KUKA KRL program: MyProgram_148().src

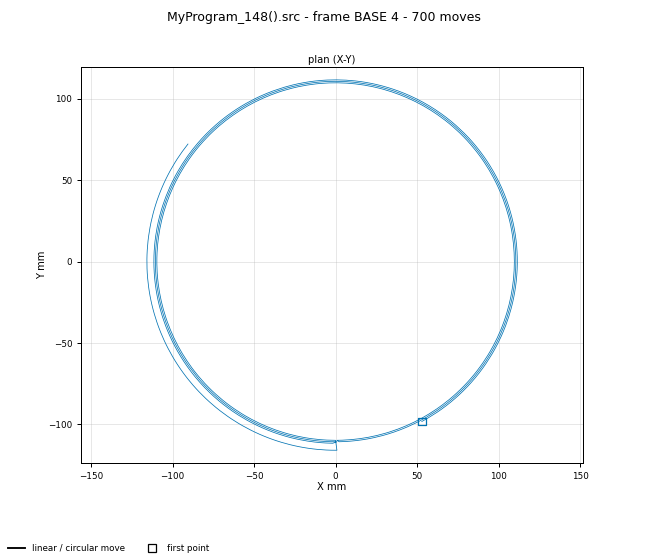
[picture p0: tool path of MyProgram_148().src in frame BASE 4, 700 of 700 moves have a stored position in this frame; points joined in program order, loops and branches not executed]
&ACCESS RVP
&REL 1
&PARAM TEMPLATE = C:\KRC\Roboter\Template\vorgabe
&PARAM EDITMASK = *
DEF MyProgram_148()
; ---- Setting reference (Base) ----
$BASE = BASE_DATA[4]

; --------------------------
; ---- Setting tool (TCP) ----
$TOOL = TOOL_DATA[3]
; --------------------------

$VEL.CP = VEL_APROX_PRINT
Startdeposition()
$VEL.CP = VEL_PRINT
LIN {X 52.9092,Y -98.1836,Z 116,A -65.1294,B 24.9503,C -1.6291,E1 25.0771,E2 510.9527} C_DIS
LIN {X 56.1114,Y -96.3909,Z 116,A -62.9664,B 24.9493,C -1.6449,E1 25.0824,E2 508.7589} C_DIS
LIN {X 62.3127,Y -92.5013,Z 116,A -59.4929,B 24.9496,C -1.6394,E1 25.0905,E2 505.3097} C_DIS
LIN {X 64.7563,Y -90.8071,Z 116,A -57.9766,B 24.9495,C -1.642,E1 25.094,E2 503.7925} C_DIS
LIN {X 67.8359,Y -88.5308,Z 116,A -55.9854,B 24.9491,C -1.6473,E1 25.0984,E2 501.7959} C_DIS
LIN {X 70.585,Y -86.3555,Z 116,A -54.1202,B 24.9487,C -1.6542,E1 25.1025,E2 499.9216} C_DIS
LIN {X 73.3349,Y -84.0315,Z 116,A -52.3931,B 24.9488,C -1.6529,E1 25.1062,E2 498.2042} C_DIS
LIN {X 75.9292,Y -81.6976,Z 116,A -50.5067,B 24.9483,C -1.6614,E1 25.1101,E2 496.3055} C_DIS
LIN {X 78.3692,Y -79.3573,Z 116,A -48.8923,B 24.9483,C -1.6601,E1 25.1133,E2 494.7009} C_DIS
LIN {X 80.9245,Y -76.7513,Z 116,A -47.0003,B 24.948,C -1.6655,E1 25.117,E2 492.8042} C_DIS
LIN {X 83.3621,Y -74.096,Z 116,A -45.0491,B 24.9474,C -1.6748,E1 25.1206,E2 490.8398} C_DIS
LIN {X 85.7734,Y -71.2898,Z 116,A -43.2959,B 24.9475,C -1.6731,E1 25.1238,E2 489.0986} C_DIS
LIN {X 87.8724,Y -68.6885,Z 116,A -41.4437,B 24.9469,C -1.6839,E1 25.127,E2 487.2296} C_DIS
LIN {X 90.2553,Y -65.5248,Z 116,A -39.4352,B 24.9466,C -1.6883,E1 25.1303,E2 485.2204} C_DIS
LIN {X 92.2402,Y -62.6984,Z 116,A -37.8546,B 24.9468,C -1.6844,E1 25.1328,E2 483.6567} C_DIS
LIN {X 95.8631,Y -57.0057,Z 116,A -34.2163,B 24.9457,C -1.7022,E1 25.1382,E2 479.9948} C_DIS
LIN {X 97.4564,Y -54.2363,Z 116,A -32.1233,B 24.9441,C -1.7278,E1 25.1412,E2 477.8523} C_DIS
LIN {X 99.4062,Y -50.5743,Z 116,A -30.4639,B 24.945,C -1.7125,E1 25.1432,E2 476.2379} C_DIS
LIN {X 101.6484,Y -45.9013,Z 116,A -27.9485,B 24.945,C -1.7138,E1 25.1462,E2 473.733} C_DIS
LIN {X 102.9872,Y -42.8163,Z 116,A -26.2004,B 24.9446,C -1.72,E1 25.1481,E2 471.9797} C_DIS
LIN {X 104.3967,Y -39.2519,Z 116,A -24.253,B 24.9442,C -1.7252,E1 25.1501,E2 470.031} C_DIS
LIN {X 105.5601,Y -36.0073,Z 116,A -22.4909,B 24.9439,C -1.7304,E1 25.1517,E2 468.2667} C_DIS
LIN {X 106.3439,Y -33.6253,Z 116,A -20.9984,B 24.943,C -1.7438,E1 25.153,E2 466.751} C_DIS
LIN {X 107.7745,Y -28.7076,Z 116,A -18.5694,B 24.943,C -1.7429,E1 25.1548,E2 464.338} C_DIS
LIN {X 108.7112,Y -24.9243,Z 116,A -16.7996,B 24.9433,C -1.7387,E1 25.1559,E2 462.5884} C_DIS
LIN {X 109.3364,Y -22.0232,Z 116,A -15.2816,B 24.943,C -1.7433,E1 25.1568,E2 461.0683} C_DIS
LIN {X 109.9232,Y -18.8799,Z 116,A -13.4529,B 24.9421,C -1.7571,E1 25.1577,E2 459.2177} C_DIS
LIN {X 110.4369,Y -15.5885,Z 116,A -11.7848,B 24.9419,C -1.7607,E1 25.1584,E2 457.551} C_DIS
LIN {X 110.8616,Y -12.2227,Z 116,A -10.0076,B 24.9414,C -1.768,E1 25.159,E2 455.7672} C_DIS
LIN {X 111.2013,Y -8.5827,Z 116,A -7.8213,B 24.9401,C -1.7883,E1 25.1595,E2 453.5459} C_DIS
LIN {X 111.4062,Y -5.3144,Z 116,A -6.3852,B 24.9405,C -1.7824,E1 25.1597,E2 452.1322} C_DIS
LIN {X 111.5251,Y -1.3818,Z 116,A -4.5343,B 24.9405,C -1.7812,E1 25.1597,E2 450.2953} C_DIS
LIN {X 111.4999,Y 2.7453,Z 116,A -1.9208,B 24.9385,C -1.8108,E1 25.1597,E2 447.6275} C_DIS
LIN {X 111.3508,Y 6.351,Z 116,A -0.5664,B 24.9397,C -1.7938,E1 25.1595,E2 446.3212} C_DIS
LIN {X 111.1521,Y 9.1985,Z 116,A 1.3678,B 24.9379,C -1.82,E1 25.159,E2 444.3366} C_DIS
LIN {X 110.7896,Y 12.8447,Z 116,A 2.7241,B 24.9391,C -1.8019,E1 25.1586,E2 443.0311} C_DIS
LIN {X 110.2953,Y 16.5677,Z 116,A 4.7378,B 24.9385,C -1.8119,E1 25.1578,E2 441.0057} C_DIS
LIN {X 109.7106,Y 20.0748,Z 116,A 6.5958,B 24.938,C -1.8191,E1 25.1569,E2 439.1416} C_DIS
LIN {X 108.9851,Y 23.6972,Z 116,A 8.3703,B 24.938,C -1.8194,E1 25.1559,E2 437.3767} C_DIS
LIN {X 108.1757,Y 27.161,Z 116,A 10.2711,B 24.9373,C -1.8284,E1 25.1546,E2 435.4655} C_DIS
LIN {X 107.3561,Y 30.2325,Z 116,A 11.7358,B 24.9375,C -1.8258,E1 25.1536,E2 434.0154} C_DIS
LIN {X 106.2715,Y 33.8515,Z 116,A 13.8167,B 24.9367,C -1.8381,E1 25.1518,E2 431.9175} C_DIS
LIN {X 105.0919,Y 37.3513,Z 116,A 16.2291,B 24.9346,C -1.8674,E1 25.1496,E2 429.4496} C_DIS
LIN {X 103.5813,Y 41.3594,Z 116,A 18.0483,B 24.9354,C -1.8564,E1 25.1477,E2 427.6663} C_DIS
LIN {X 101.9341,Y 45.2672,Z 116,A 20.0203,B 24.9356,C -1.8533,E1 25.1455,E2 425.7125} C_DIS
LIN {X 100.5925,Y 48.1713,Z 116,A 21.698,B 24.9352,C -1.8596,E1 25.1435,E2 424.029} C_DIS
LIN {X 98.7423,Y 51.8584,Z 116,A 23.6261,B 24.9354,C -1.8568,E1 25.1411,E2 422.1176} C_DIS
LIN {X 97.0537,Y 54.9566,Z 116,A 25.6699,B 24.9343,C -1.8722,E1 25.1383,E2 420.0482} C_DIS
LIN {X 94.5285,Y 59.1919,Z 116,A 28.0302,B 24.9343,C -1.8712,E1 25.1349,E2 417.7022} C_DIS
LIN {X 92.7016,Y 62.017,Z 116,A 29.8036,B 24.9339,C -1.8777,E1 25.1322,E2 415.9223} C_DIS
LIN {X 91.0092,Y 64.473,Z 116,A 31.3362,B 24.9336,C -1.8816,E1 25.1297,E2 414.388} C_DIS
LIN {X 88.7627,Y 67.5349,Z 116,A 33.5767,B 24.9324,C -1.8994,E1 25.1259,E2 412.1161} C_DIS
LIN {X 85.9589,Y 71.0665,Z 116,A 35.5596,B 24.933,C -1.89,E1 25.1225,E2 410.1646} C_DIS
LIN {X 83.7079,Y 73.7055,Z 116,A 37.3159,B 24.9328,C -1.893,E1 25.1192,E2 408.4092} C_DIS
LIN {X 81.6754,Y 75.9528,Z 116,A 39.3987,B 24.9309,C -1.9201,E1 25.1152,E2 406.2717} C_DIS
LIN {X 78.9056,Y 78.8264,Z 116,A 40.8065,B 24.9326,C -1.8958,E1 25.1125,E2 404.9272} C_DIS
LIN {X 73.6893,Y 83.722,Z 116,A 44.6367,B 24.9316,C -1.9102,E1 25.1047,E2 401.0785} C_DIS
LIN {X 70.7104,Y 86.2539,Z 116,A 46.6082,B 24.9314,C -1.9124,E1 25.1004,E2 399.1093} C_DIS
LIN {X 67.7988,Y 88.5593,Z 116,A 48.5399,B 24.9311,C -1.917,E1 25.0962,E2 397.174} C_DIS
LIN {X 64.6194,Y 90.9048,Z 116,A 50.7894,B 24.9302,C -1.9302,E1 25.091,E2 394.9011} C_DIS
LIN {X 60.8841,Y 93.4495,Z 116,A 52.8224,B 24.9308,C -1.9213,E1 25.0863,E2 392.896} C_DIS
LIN {X 57.336,Y 95.668,Z 116,A 55.1632,B 24.93,C -1.9329,E1 25.0807,E2 390.535} C_DIS
LIN {X 53.72,Y 97.7434,Z 116,A 57.238,B 24.93,C -1.933,E1 25.0757,E2 388.4661} C_DIS
LIN {X 49.7844,Y 99.8043,Z 116,A 59.6973,B 24.9292,C -1.9437,E1 25.0695,E2 385.9882} C_DIS
LIN {X 45.4869,Y 101.8351,Z 116,A 61.7418,B 24.9302,C -1.9293,E1 25.0644,E2 383.9829} C_DIS
LIN {X 42.4471,Y 103.1394,Z 116,A 63.4921,B 24.9299,C -1.9333,E1 25.0599,E2 382.2272} C_DIS
LIN {X 38.7978,Y 104.5678,Z 116,A 65.399,B 24.9301,C -1.9307,E1 25.055,E2 380.3308} C_DIS
LIN {X 35.1737,Y 105.8412,Z 116,A 67.4613,B 24.9297,C -1.9362,E1 25.0495,E2 378.2594} C_DIS
LIN {X 32.2727,Y 106.7609,Z 116,A 69.4841,B 24.9282,C -1.9572,E1 25.044,E2 376.1905} C_DIS
LIN {X 28.7542,Y 107.7619,Z 116,A 70.8582,B 24.9297,C -1.9368,E1 25.0404,E2 374.867} C_DIS
LIN {X 25.1913,Y 108.6495,Z 116,A 72.7621,B 24.9295,C -1.9386,E1 25.0352,E2 372.9615} C_DIS
LIN {X 22.2287,Y 109.2943,Z 116,A 74.4419,B 24.9291,C -1.9445,E1 25.0306,E2 371.2699} C_DIS
LIN {X 18.5918,Y 109.9713,Z 116,A 76.155,B 24.9296,C -1.9373,E1 25.0259,E2 369.5757} C_DIS
LIN {X 15.9494,Y 110.3857,Z 116,A 77.5464,B 24.9296,C -1.9384,E1 25.0221,E2 368.183} C_DIS
LIN {X 12.0058,Y 110.8843,Z 116,A 79.7842,B 24.9289,C -1.947,E1 25.0158,E2 365.9263} C_DIS
LIN {X 6.4381,Y 111.346,Z 116,A 82.5158,B 24.9293,C -1.9413,E1 25.0083,E2 363.2096} C_DIS
LIN {X 3.0813,Y 111.4896,Z 116,A 84.2013,B 24.9295,C -1.9395,E1 25.0036,E2 361.5289} C_DIS
LIN {X 0.6202,Y 111.5299,Z 116,A 85.7304,B 24.9287,C -1.9504,E1 24.9992,E2 359.9741} C_DIS
LIN {X -5.1396,Y 111.4137,Z 116,A 88.4976,B 24.9293,C -1.9414,E1 24.9916,E2 357.2277} C_DIS
LIN {X -8.4005,Y 111.216,Z 116,A 90.2558,B 24.9291,C -1.9441,E1 24.9867,E2 355.4626} C_DIS
LIN {X -12.4768,Y 110.8327,Z 116,A 92.6726,B 24.9283,C -1.956,E1 24.9799,E2 353.0162} C_DIS
LIN {X -15.8136,Y 110.405,Z 116,A 93.9929,B 24.9296,C -1.9379,E1 24.9763,E2 351.7375} C_DIS
LIN {X -19.4553,Y 109.8221,Z 116,A 95.9142,B 24.9296,C -1.9377,E1 24.971,E2 349.8151} C_DIS
LIN {X -23.038,Y 109.1281,Z 116,A 97.8293,B 24.9296,C -1.9377,E1 24.9658,E2 347.8977} C_DIS
LIN {X -26.4229,Y 108.3565,Z 116,A 99.5348,B 24.93,C -1.9329,E1 24.9612,E2 346.2014} C_DIS
LIN {X -29.291,Y 107.6169,Z 116,A 101.0996,B 24.93,C -1.9331,E1 24.9569,E2 344.6337} C_DIS
LIN {X -31.5254,Y 106.9836,Z 116,A 103.5992,B 24.9261,C -1.9857,E1 24.95,E2 342.0049} C_DIS
LIN {X -38.4898,Y 104.6801,Z 116,A 106.5973,B 24.9288,C -1.9489,E1 24.9423,E2 339.0881} C_DIS
LIN {X -42.1959,Y 103.2417,Z 116,A 108.6809,B 24.9288,C -1.9477,E1 24.9369,E2 337.0027} C_DIS
LIN {X -46.0009,Y 101.6034,Z 116,A 110.2767,B 24.9307,C -1.9229,E1 24.9329,E2 335.4621} C_DIS
LIN {X -49.297,Y 100.0459,Z 116,A 112.1442,B 24.9309,C -1.9197,E1 24.9283,E2 333.5974} C_DIS
LIN {X -54.9445,Y 97.061,Z 116,A 115.5039,B 24.9311,C -1.9172,E1 24.92,E2 330.2342} C_DIS
LIN {X -57.6585,Y 95.472,Z 116,A 117.0868,B 24.9314,C -1.9129,E1 24.9162,E2 328.6566} C_DIS
LIN {X -60.6647,Y 93.5914,Z 116,A 118.9691,B 24.9314,C -1.9118,E1 24.9118,E2 326.7708} C_DIS
LIN {X -63.5165,Y 91.6788,Z 116,A 120.8591,B 24.9314,C -1.9134,E1 24.9074,E2 324.8708} C_DIS
LIN {X -66.9482,Y 89.2034,Z 116,A 123.5372,B 24.9302,C -1.929,E1 24.9013,E2 322.1459} C_DIS
LIN {X -70.7502,Y 86.2217,Z 116,A 125.8474,B 24.9311,C -1.9166,E1 24.8964,E2 319.8565} C_DIS
LIN {X -73.7129,Y 83.7014,Z 116,A 127.3539,B 24.9329,C -1.8925,E1 24.8933,E2 318.4015} C_DIS
LIN {X -76.5079,Y 81.1534,Z 116,A 129.8759,B 24.9315,C -1.9109,E1 24.888,E2 315.8252} C_DIS
LIN {X -79.5478,Y 78.1763,Z 116,A 132.0811,B 24.9319,C -1.9063,E1 24.8837,E2 313.6216} C_DIS
LIN {X -82.5085,Y 75.0459,Z 116,A 133.7954,B 24.9337,C -1.8809,E1 24.8806,E2 311.9602} C_DIS
LIN {X -84.5818,Y 72.7012,Z 116,A 135.9859,B 24.9323,C -1.8998,E1 24.8765,E2 309.7147} C_DIS
LIN {X -87.4363,Y 69.2402,Z 116,A 137.8303,B 24.9341,C -1.8755,E1 24.8734,E2 307.9197} C_DIS
LIN {X -90.8086,Y 64.7542,Z 116,A 140.4061,B 24.9355,C -1.8556,E1 24.8692,E2 305.3789} C_DIS
LIN {X -94.0747,Y 59.9117,Z 116,A 143.6719,B 24.9353,C -1.8574,E1 24.8641,E2 302.0924} C_DIS
LIN {X -96.813,Y 55.3769,Z 116,A 146.2308,B 24.9363,C -1.8432,E1 24.8605,E2 299.5542} C_DIS
LIN {X -98.3015,Y 52.6919,Z 116,A 147.9315,B 24.9363,C -1.8434,E1 24.8582,E2 297.8441} C_DIS
LIN {X -100.3136,Y 48.7518,Z 116,A 150.216,B 24.9367,C -1.837,E1 24.8554,E2 295.5625} C_DIS
LIN {X -101.6068,Y 45.9935,Z 116,A 151.6526,B 24.9374,C -1.8273,E1 24.8537,E2 294.1411} C_DIS
LIN {X -104.1686,Y 39.8541,Z 116,A 155.2238,B 24.9377,C -1.8227,E1 24.8499,E2 290.5611} C_DIS
LIN {X -105.2317,Y 36.9541,Z 116,A 156.6956,B 24.9384,C -1.8133,E1 24.8485,E2 289.1033} C_DIS
LIN {X -106.0707,Y 34.4723,Z 116,A 158.7014,B 24.9369,C -1.8347,E1 24.8468,E2 287.0348} C_DIS
LIN {X -107.263,Y 30.561,Z 116,A 159.9553,B 24.9396,C -1.7952,E1 24.8459,E2 285.8681} C_DIS
LIN {X -108.04,Y 27.6889,Z 116,A 162.1523,B 24.9382,C -1.8162,E1 24.8443,E2 283.6082} C_DIS
LIN {X -108.826,Y 24.4269,Z 116,A 163.447,B 24.9397,C -1.794,E1 24.8435,E2 282.3589} C_DIS
LIN {X -109.5487,Y 20.9374,Z 116,A 166.1596,B 24.9377,C -1.8225,E1 24.842,E2 279.5622} C_DIS
LIN {X -110.3857,Y 15.9494,Z 116,A 168.0257,B 24.9403,C -1.7854,E1 24.8413,E2 277.7733} C_DIS
LIN {X -110.8645,Y 12.1948,Z 116,A 170.0214,B 24.9405,C -1.7811,E1 24.8406,E2 275.7761} C_DIS
LIN {X -111.1664,Y 9.0196,Z 116,A 171.5106,B 24.9413,C -1.77,E1 24.8402,E2 274.3043} C_DIS
LIN {X -111.3505,Y 6.3572,Z 116,A 172.8897,B 24.9416,C -1.7659,E1 24.84,E2 272.9268} C_DIS
LIN {X -111.4802,Y 3.3861,Z 116,A 174.5077,B 24.9416,C -1.7644,E1 24.8398,E2 271.3026} C_DIS
LIN {X -111.5316,Y -0.2035,Z 116,A 176.3564,B 24.942,C -1.7586,E1 24.8398,E2 269.4566} C_DIS
LIN {X -111.4807,Y -3.3722,Z 116,A 178.0458,B 24.9422,C -1.7557,E1 24.8399,E2 267.7639} C_DIS
LIN {X -111.3074,Y -7.0828,Z 116,A -179.9817,B 24.9425,C -1.752,E1 24.8402,E2 265.7883} C_DIS
LIN {X -110.9839,Y -11.0543,Z 116,A -178.0528,B 24.9432,C -1.7408,E1 24.8407,E2 263.8745} C_DIS
LIN {X -110.6319,Y -14.1394,Z 116,A -176.3798,B 24.9433,C -1.7388,E1 24.8413,E2 262.1964} C_DIS
LIN {X -110.1255,Y -17.6658,Z 116,A -174.4928,B 24.9436,C -1.7352,E1 24.8421,E2 260.3068} C_DIS
LIN {X -109.5137,Y -21.12,Z 116,A -172.7188,B 24.944,C -1.7284,E1 24.843,E2 258.5384} C_DIS
LIN {X -108.9187,Y -24.0018,Z 116,A -170.7974,B 24.9433,C -1.7397,E1 24.8441,E2 256.5787} C_DIS
LIN {X -108.1112,Y -27.4119,Z 116,A -169.4795,B 24.9449,C -1.7153,E1 24.845,E2 255.3114} C_DIS
LIN {X -106.7177,Y -32.4191,Z 116,A -166.7876,B 24.9453,C -1.7079,E1 24.8471,E2 252.6215} C_DIS
LIN {X -105.8504,Y -35.1463,Z 116,A -165.3312,B 24.9457,C -1.7029,E1 24.8483,E2 251.1686} C_DIS
LIN {X -104.284,Y -39.5494,Z 116,A -162.8738,B 24.946,C -1.698,E1 24.8507,E2 248.7091} C_DIS
LIN {X -103.0393,Y -42.6919,Z 116,A -161.0095,B 24.946,C -1.698,E1 24.8526,E2 246.8346} C_DIS
LIN {X -101.7991,Y -45.5668,Z 116,A -159.4265,B 24.9463,C -1.6923,E1 24.8544,E2 245.2562} C_DIS
LIN {X -100.3926,Y -48.5875,Z 116,A -157.7871,B 24.9468,C -1.6846,E1 24.8563,E2 243.6263} C_DIS
LIN {X -98.5083,Y -52.3026,Z 116,A -155.6007,B 24.9471,C -1.6805,E1 24.8592,E2 241.4381} C_DIS
LIN {X -97.1042,Y -54.8671,Z 116,A -153.8534,B 24.9467,C -1.6861,E1 24.8616,E2 239.6682} C_DIS
LIN {X -94.9548,Y -58.5095,Z 116,A -151.8064,B 24.9474,C -1.6753,E1 24.8645,E2 237.6364} C_DIS
LIN {X -93.0405,Y -61.5044,Z 116,A -150.0365,B 24.9478,C -1.6683,E1 24.8672,E2 235.8742} C_DIS
LIN {X -90.9636,Y -64.537,Z 116,A -148.186,B 24.9482,C -1.662,E1 24.8701,E2 234.0296} C_DIS
LIN {X -88.3938,Y -68.0134,Z 116,A -145.5244,B 24.9475,C -1.6742,E1 24.8747,E2 231.3262} C_DIS
LIN {X -86.2167,Y -70.7563,Z 116,A -144.0253,B 24.9485,C -1.6579,E1 24.8773,E2 229.8591} C_DIS
LIN {X -83.5848,Y -73.8464,Z 116,A -141.7264,B 24.9483,C -1.6617,E1 24.8815,E2 227.5407} C_DIS
LIN {X -80.3251,Y -77.3769,Z 116,A -139.5713,B 24.9494,C -1.6436,E1 24.8856,E2 225.4192} C_DIS
LIN {X -77.0941,Y -80.5977,Z 116,A -137.0655,B 24.9493,C -1.6452,E1 24.8906,E2 222.8991} C_DIS
LIN {X -74.3744,Y -83.1129,Z 116,A -135.3031,B 24.9499,C -1.6357,E1 24.8942,E2 221.1523} C_DIS
LIN {X -71.6856,Y -85.4445,Z 116,A -133.3821,B 24.9499,C -1.6359,E1 24.8983,E2 219.2234} C_DIS
LIN {X -69.227,Y -87.4468,Z 116,A -131.7489,B 24.95,C -1.6331,E1 24.9019,E2 217.5908} C_DIS
LIN {X -65.9884,Y -89.9158,Z 116,A -129.6715,B 24.9503,C -1.6288,E1 24.9065,E2 215.5162} C_DIS
LIN {X -63.0004,Y -92.0357,Z 116,A -127.7385,B 24.9503,C -1.6277,E1 24.911,E2 213.5792} C_DIS
LIN {X -59.5862,Y -94.2822,Z 116,A -125.4209,B 24.95,C -1.6333,E1 24.9165,E2 211.2407} C_DIS
LIN {X -54.3465,Y -97.3949,Z 116,A -122.5967,B 24.9511,C -1.6162,E1 24.9232,E2 208.4487} C_DIS
LIN {X -52.1961,Y -98.5644,Z 116,A -120.9552,B 24.9502,C -1.6304,E1 24.9273,E2 206.7689} C_DIS
LIN {X -48.1302,Y -100.6122,Z 116,A -118.9814,B 24.9513,C -1.6124,E1 24.9322,E2 204.8326} C_DIS
LIN {X -45.0177,Y -102.0439,Z 116,A -117.1605,B 24.9513,C -1.613,E1 24.9368,E2 203.0062} C_DIS
LIN {X -41.9734,Y -103.3322,Z 116,A -115.5832,B 24.9517,C -1.6062,E1 24.9409,E2 201.4413} C_DIS
LIN {X -38.2833,Y -104.7554,Z 116,A -113.4849,B 24.9517,C -1.6071,E1 24.9464,E2 199.3366} C_DIS
LIN {X -35.4239,Y -105.7568,Z 116,A -111.5717,B 24.9508,C -1.6207,E1 24.9515,E2 197.3873} C_DIS
LIN {X -30.6504,Y -107.2377,Z 116,A -109.3204,B 24.9517,C -1.6056,E1 24.9575,E2 195.1681} C_DIS
LIN {X -27.1861,Y -108.1692,Z 116,A -107.5707,B 24.952,C -1.6006,E1 24.9622,E2 193.4278} C_DIS
LIN {X -23.0365,Y -109.1284,Z 116,A -105.2378,B 24.9517,C -1.6056,E1 24.9686,E2 191.08} C_DIS
LIN {X -19.6611,Y -109.7851,Z 116,A -103.5339,B 24.9519,C -1.6024,E1 24.9732,E2 189.3821} C_DIS
LIN {X -17.1552,Y -110.2044,Z 116,A -102.0814,B 24.9515,C -1.6082,E1 24.9773,E2 187.9142} C_DIS
LIN {X -12.8611,Y -110.7877,Z 116,A -99.4591,B 24.9505,C -1.6248,E1 24.9847,E2 185.251} C_DIS
LIN {X -8.9519,Y -111.1718,Z 116,A -97.9302,B 24.9518,C -1.6037,E1 24.9888,E2 183.7712} C_DIS
LIN {X -6.097,Y -111.3649,Z 116,A -96.224,B 24.9512,C -1.6139,E1 24.9936,E2 182.0404} C_DIS
LIN {X -1.7181,Y -111.5189,Z 116,A -93.6675,B 24.9504,C -1.6275,E1 25.0009,E2 179.4515} C_DIS
LIN {X -1.7181,Y -111.5189,Z 116,A -93.6675,B 24.9504,C -1.6275,E1 25.0009,E2 179.4515} C_DIS
Enddeposition()
LIN {X 0.7946,Y -110.6158,Z 116,A -93.2714,B 24.9517,C -1.6052,E1 25.0018,E2 179.1083} C_DIS
Startdeposition()
$VEL.CP = VEL_PRINT
LIN {X -2.6442,Y -110.5946,Z 116,A -95.4467,B 24.9527,C -1.5881,E1 24.9956,E2 181.3241} C_DIS
LIN {X -6.5349,Y -110.4321,Z 116,A -97.5104,B 24.9529,C -1.586,E1 24.9898,E2 183.3933} C_DIS
LIN {X -9.5144,Y -110.2165,Z 116,A -99.3021,B 24.9535,C -1.5759,E1 24.9848,E2 185.2098} C_DIS
LIN {X -12.7964,Y -109.8819,Z 116,A -100.7721,B 24.9529,C -1.586,E1 24.9808,E2 186.6567} C_DIS
LIN {X -15.973,Y -109.466,Z 116,A -102.4709,B 24.9529,C -1.5847,E1 24.9761,E2 188.3599} C_DIS
LIN {X -19.2037,Y -108.9456,Z 116,A -103.9916,B 24.9525,C -1.5924,E1 24.9719,E2 189.8637} C_DIS
LIN {X -21.3846,Y -108.539,Z 116,A -105.2338,B 24.9527,C -1.589,E1 24.9685,E2 191.1153} C_DIS
LIN {X -23.5267,Y -108.0938,Z 116,A -106.4605,B 24.9529,C -1.5857,E1 24.9651,E2 192.3515} C_DIS
LIN {X -26.055,Y -107.5125,Z 116,A -107.7487,B 24.9527,C -1.5887,E1 24.9616,E2 193.6343} C_DIS
LIN {X -29.519,Y -106.6154,Z 116,A -109.5858,B 24.9527,C -1.5904,E1 24.9567,E2 195.47} C_DIS
LIN {X -31.9801,Y -105.9025,Z 116,A -111.4499,B 24.9538,C -1.5696,E1 24.9515,E2 197.3869} C_DIS
LIN {X -35.3248,Y -104.8329,Z 116,A -112.8332,B 24.9527,C -1.5887,E1 24.948,E2 198.7273} C_DIS
LIN {X -39.5172,Y -103.3262,Z 116,A -115.1086,B 24.9525,C -1.5921,E1 24.942,E2 200.9993} C_DIS
LIN {X -42.1139,Y -102.2956,Z 116,A -116.4787,B 24.9522,C -1.5966,E1 24.9385,E2 202.3616} C_DIS
LIN {X -45.0316,Y -101.0453,Z 116,A -118.0904,B 24.952,C -1.5997,E1 24.9344,E2 203.9697} C_DIS
LIN {X -47.1371,Y -100.0806,Z 116,A -119.3351,B 24.952,C -1.5993,E1 24.9312,E2 205.2186} C_DIS
LIN {X -49.1035,Y -99.1293,Z 116,A -120.4083,B 24.9519,C -1.603,E1 24.9285,E2 206.2857} C_DIS
LIN {X -52.1502,Y -97.5633,Z 116,A -122.269,B 24.9519,C -1.6018,E1 24.9239,E2 208.1544} C_DIS
LIN {X -55.258,Y -95.835,Z 116,A -124.1893,B 24.9519,C -1.6013,E1 24.9192,E2 210.0816} C_DIS
LIN {X -58.5749,Y -93.8444,Z 116,A -126.2251,B 24.9519,C -1.603,E1 24.9144,E2 212.1196} C_DIS
LIN {X -61.4116,Y -92.0151,Z 116,A -127.8814,B 24.9515,C -1.6094,E1 24.9105,E2 213.7661} C_DIS
LIN {X -64.1862,Y -90.0995,Z 116,A -129.7428,B 24.9515,C -1.6078,E1 24.9062,E2 215.6377} C_DIS
LIN {X -67.0583,Y -87.9847,Z 116,A -131.6136,B 24.9515,C -1.6101,E1 24.9021,E2 217.5097} C_DIS
LIN {X -69.7861,Y -85.8354,Z 116,A -133.3515,B 24.9511,C -1.6158,E1 24.8983,E2 219.2404} C_DIS
LIN {X -72.77,Y -83.3205,Z 116,A -135.3311,B 24.9507,C -1.6214,E1 24.8941,E2 221.2145} C_DIS
LIN {X -75.0304,Y -81.2916,Z 116,A -136.9337,B 24.9507,C -1.6234,E1 24.8908,E2 222.8188} C_DIS
LIN {X -77.8122,Y -78.6324,Z 116,A -138.945,B 24.9504,C -1.6269,E1 24.8867,E2 224.8301} C_DIS
LIN {X -80.025,Y -76.3811,Z 116,A -140.7607,B 24.9506,C -1.6233,E1 24.8832,E2 226.6621} C_DIS
LIN {X -82.6641,Y -73.5157,Z 116,A -142.5618,B 24.9498,C -1.6363,E1 24.8799,E2 228.4403} C_DIS
LIN {X -84.5753,Y -71.3101,Z 116,A -144.2654,B 24.9501,C -1.6323,E1 24.8767,E2 230.1611} C_DIS
LIN {X -89.8204,Y -64.5774,Z 116,A -148.4081,B 24.9487,C -1.6539,E1 24.8698,E2 234.2722} C_DIS
LIN {X -91.7647,Y -61.7827,Z 116,A -150.2724,B 24.9487,C -1.6544,E1 24.8668,E2 236.1443} C_DIS
LIN {X -93.4706,Y -59.1732,Z 116,A -151.9311,B 24.9486,C -1.6569,E1 24.8643,E2 237.8055} C_DIS
LIN {X -94.9201,Y -56.8183,Z 116,A -153.5828,B 24.9488,C -1.6523,E1 24.8618,E2 239.4767} C_DIS
LIN {X -96.9005,Y -53.3712,Z 116,A -155.6331,B 24.9485,C -1.6582,E1 24.859,E2 241.5237} C_DIS
LIN {X -98.55,Y -50.2563,Z 116,A -157.413,B 24.948,C -1.6651,E1 24.8568,E2 243.2968} C_DIS
LIN {X -100.3145,Y -46.6345,Z 116,A -159.4848,B 24.9476,C -1.6716,E1 24.8543,E2 245.3644} C_DIS
LIN {X -101.589,Y -43.7911,Z 116,A -160.9886,B 24.9471,C -1.6804,E1 24.8526,E2 246.8554} C_DIS
LIN {X -102.6665,Y -41.2027,Z 116,A -162.6467,B 24.9473,C -1.6768,E1 24.8508,E2 248.5314} C_DIS
LIN {X -104.1452,Y -37.309,Z 116,A -164.8304,B 24.947,C -1.6821,E1 24.8487,E2 250.7145} C_DIS
LIN {X -105.4494,Y -33.4457,Z 116,A -166.7619,B 24.9461,C -1.6954,E1 24.847,E2 252.6255} C_DIS
LIN {X -106.7136,Y -29.1561,Z 116,A -169.2007,B 24.946,C -1.6978,E1 24.8452,E2 255.0727} C_DIS
LIN {X -107.5482,Y -25.9087,Z 116,A -171.1503,B 24.9462,C -1.6951,E1 24.8438,E2 257.0401} C_DIS
LIN {X -108.4813,Y -21.6779,Z 116,A -173.3381,B 24.9456,C -1.7043,E1 24.8426,E2 259.219} C_DIS
LIN {X -109.2258,Y -17.5477,Z 116,A -175.2833,B 24.9446,C -1.7198,E1 24.8417,E2 261.1388} C_DIS
LIN {X -109.557,Y -15.3326,Z 116,A -176.4591,B 24.9444,C -1.7229,E1 24.8412,E2 262.3141} C_DIS
LIN {X -109.9712,Y -12.0151,Z 116,A -178.3434,B 24.9444,C -1.7226,E1 24.8406,E2 264.2103} C_DIS
LIN {X -110.2825,Y -8.6922,Z 116,A 179.9375,B 24.944,C -1.7286,E1 24.8402,E2 265.9256} C_DIS
LIN {X -110.4869,Y -5.5449,Z 116,A 178.4055,B 24.9434,C -1.7376,E1 24.8399,E2 267.4451} C_DIS
LIN {X -110.6035,Y -2.1578,Z 116,A 176.5375,B 24.9434,C -1.7391,E1 24.8398,E2 269.321} C_DIS
LIN {X -110.6116,Y 1.7189,Z 116,A 174.537,B 24.9429,C -1.7459,E1 24.8398,E2 271.3173} C_DIS
LIN {X -110.5029,Y 5.2045,Z 116,A 172.8221,B 24.9423,C -1.7552,E1 24.84,E2 273.0204} C_DIS
LIN {X -110.359,Y 7.6624,Z 116,A 171.3894,B 24.9423,C -1.7534,E1 24.8403,E2 274.4659} C_DIS
LIN {X -110.0288,Y 11.4645,Z 116,A 169.4518,B 24.9419,C -1.7613,E1 24.8408,E2 276.3963} C_DIS
LIN {X -109.5688,Y 15.2496,Z 116,A 166.3322,B 24.9442,C -1.725,E1 24.842,E2 279.6211} C_DIS
LIN {X -108.4938,Y 21.617,Z 116,A 164.1829,B 24.9406,C -1.7803,E1 24.8431,E2 281.6512} C_DIS
LIN {X -107.8858,Y 24.467,Z 116,A 162.0703,B 24.9418,C -1.7625,E1 24.8444,E2 283.8187} C_DIS
LIN {X -106.9715,Y 28.2015,Z 116,A 160.6439,B 24.9399,C -1.79,E1 24.8453,E2 285.1877} C_DIS
LIN {X -105.5341,Y 33.1742,Z 116,A 157.9865,B 24.9393,C -1.7995,E1 24.8474,E2 287.8381} C_DIS
LIN {X -104.5999,Y 36.0147,Z 116,A 156.2336,B 24.9395,C -1.7966,E1 24.849,E2 289.6078} C_DIS
LIN {X -103.2432,Y 39.7363,Z 116,A 154.1729,B 24.9391,C -1.8026,E1 24.851,E2 291.6657} C_DIS
LIN {X -101.5884,Y 43.7924,Z 116,A 152.1388,B 24.938,C -1.8185,E1 24.8532,E2 293.6732} C_DIS
LIN {X -100.4942,Y 46.2484,Z 116,A 150.4967,B 24.9384,C -1.8133,E1 24.8551,E2 295.3369} C_DIS
LIN {X -98.822,Y 49.7236,Z 116,A 148.3895,B 24.9382,C -1.8151,E1 24.8577,E2 297.4511} C_DIS
LIN {X -96.8267,Y 53.5033,Z 116,A 146.4794,B 24.937,C -1.8331,E1 24.8602,E2 299.3282} C_DIS
LIN {X -95.8824,Y 55.1757,Z 116,A 145.326,B 24.9372,C -1.83,E1 24.8618,E2 300.495} C_DIS
LIN {X -93.0955,Y 59.758,Z 116,A 142.8311,B 24.9359,C -1.8488,E1 24.8654,E2 302.958} C_DIS
LIN {X -91.647,Y 61.9565,Z 116,A 141.2159,B 24.9363,C -1.843,E1 24.8679,E2 304.5952} C_DIS
LIN {X -90.0404,Y 64.269,Z 116,A 139.0083,B 24.938,C -1.8186,E1 24.8716,E2 306.8716} C_DIS
LIN {X -87.3152,Y 67.9271,Z 116,A 137.3178,B 24.9358,C -1.8504,E1 24.8744,E2 308.4944} C_DIS
LIN {X -83.4721,Y 72.5964,Z 116,A 134.4396,B 24.9346,C -1.8684,E1 24.8795,E2 311.343} C_DIS
LIN {X -79.0901,Y 77.3489,Z 116,A 129.9716,B 24.937,C -1.834,E1 24.8882,E2 315.9125} C_DIS
LIN {X -75.4466,Y 80.9062,Z 116,A 128.2004,B 24.9342,C -1.8733,E1 24.8916,E2 317.5974} C_DIS
LIN {X -70.4463,Y 85.2949,Z 116,A 124.3381,B 24.9348,C -1.865,E1 24.8999,E2 321.4943} C_DIS
LIN {X -65.9354,Y 88.8296,Z 116,A 121.2904,B 24.9346,C -1.8682,E1 24.9067,E2 324.5454} C_DIS
LIN {X -63.2972,Y 90.7264,Z 116,A 120.172,B 24.9328,C -1.8935,E1 24.9091,E2 325.6074} C_DIS
LIN {X -60.8772,Y 92.3674,Z 116,A 118.4654,B 24.9331,C -1.889,E1 24.9131,E2 327.3304} C_DIS
LIN {X -58.4459,Y 93.9249,Z 116,A 116.9407,B 24.933,C -1.8907,E1 24.9167,E2 328.856} C_DIS
LIN {X -55.0438,Y 95.9582,Z 116,A 114.9108,B 24.9327,C -1.8953,E1 24.9216,E2 330.8809} C_DIS
LIN {X -51.2917,Y 98.0154,Z 116,A 112.8086,B 24.9321,C -1.9036,E1 24.9267,E2 332.9694} C_DIS
LIN {X -48.5101,Y 99.4233,Z 116,A 111.1536,B 24.932,C -1.9046,E1 24.9308,E2 334.6265} C_DIS
LIN {X -46.0536,Y 100.5847,Z 116,A 108.9137,B 24.9342,C -1.8742,E1 24.9367,E2 336.9442} C_DIS
LIN {X -41.711,Y 102.4596,Z 116,A 107.5962,B 24.9307,C -1.9222,E1 24.9399,E2 338.1505} C_DIS
LIN {X -39.5776,Y 103.3033,Z 116,A 105.9649,B 24.9319,C -1.9062,E1 24.9442,E2 339.8233} C_DIS
LIN {X -34.6704,Y 105.0516,Z 116,A 102.9692,B 24.9325,C -1.8979,E1 24.9522,E2 342.8447} C_DIS
LIN {X -29.2761,Y 106.6812,Z 116,A 100.5666,B 24.9308,C -1.9216,E1 24.9585,E2 345.1949} C_DIS
LIN {X -26.3675,Y 107.4363,Z 116,A 98.884,B 24.931,C -1.9181,E1 24.963,E2 346.8883} C_DIS
LIN {X -23.4553,Y 108.1094,Z 116,A 97.3098,B 24.931,C -1.9184,E1 24.9673,E2 348.4637} C_DIS
LIN {X -20.8527,Y 108.6414,Z 116,A 95.9727,B 24.9308,C -1.9211,E1 24.971,E2 349.7959} C_DIS
LIN {X -17.5603,Y 109.2239,Z 116,A 94.2367,B 24.9308,C -1.9222,E1 24.9758,E2 351.5311} C_DIS
LIN {X -13.6053,Y 109.7864,Z 116,A 91.9483,B 24.9313,C -1.9146,E1 24.9821,E2 353.8391} C_DIS
LIN {X -9.5612,Y 110.2122,Z 116,A 90.0651,B 24.9306,C -1.9247,E1 24.9873,E2 355.6994} C_DIS
LIN {X -6.5104,Y 110.4335,Z 116,A 88.3784,B 24.9308,C -1.9212,E1 24.992,E2 357.395} C_DIS
LIN {X -3.006,Y 110.5843,Z 116,A 86.545,B 24.9308,C -1.9211,E1 24.9972,E2 359.2289} C_DIS
LIN {X -0.2802,Y 110.6249,Z 116,A 85.1309,B 24.9308,C -1.9213,E1 25.0011,E2 360.6425} C_DIS
LIN {X 3.1623,Y 110.5795,Z 116,A 83.2783,B 24.931,C -1.9187,E1 25.0063,E2 362.501} C_DIS
LIN {X 6.9926,Y 110.4043,Z 116,A 81.3058,B 24.931,C -1.9193,E1 25.0118,E2 364.4714} C_DIS
LIN {X 11.0021,Y 110.0773,Z 116,A 79.4557,B 24.9303,C -1.9287,E1 25.0169,E2 366.2981} C_DIS
LIN {X 14.1649,Y 109.7139,Z 116,A 77.6114,B 24.9309,C -1.9203,E1 25.022,E2 368.1609} C_DIS
LIN {X 17.3527,Y 109.256,Z 116,A 76.0891,B 24.9305,C -1.9258,E1 25.0262,E2 369.6687} C_DIS
LIN {X 19.7772,Y 108.8425,Z 116,A 74.6396,B 24.931,C -1.9181,E1 25.0302,E2 371.1349} C_DIS
LIN {X 23.7373,Y 108.0479,Z 116,A 72.6248,B 24.9309,C -1.9203,E1 25.0357,E2 373.142} C_DIS
LIN {X 26.6627,Y 107.3643,Z 116,A 71.102,B 24.9309,C -1.9208,E1 25.0398,E2 374.6615} C_DIS
LIN {X 32.1205,Y 105.8607,Z 116,A 68.1593,B 24.931,C -1.9183,E1 25.0478,E2 377.6052} C_DIS
LIN {X 36.0617,Y 104.5834,Z 116,A 66.06,B 24.931,C -1.9184,E1 25.0533,E2 379.7001} C_DIS
LIN {X 38.6032,Y 103.6723,Z 116,A 64.7124,B 24.931,C -1.9193,E1 25.0568,E2 381.0429} C_DIS
LIN {X 40.6005,Y 102.9048,Z 116,A 63.5215,B 24.9313,C -1.9147,E1 25.0599,E2 382.242} C_DIS
LIN {X 43.5913,Y 101.6761,Z 116,A 61.9088,B 24.9313,C -1.9155,E1 25.0641,E2 383.8491} C_DIS
LIN {X 45.586,Y 100.7954,Z 116,A 60.6139,B 24.9318,C -1.9072,E1 25.0674,E2 385.1603} C_DIS
LIN {X 48.9503,Y 99.2053,Z 116,A 59.0717,B 24.9308,C -1.9212,E1 25.0712,E2 386.6654} C_DIS
LIN {X 51.077,Y 98.1285,Z 116,A 57.2285,B 24.9328,C -1.8938,E1 25.0759,E2 388.5685} C_DIS
LIN {X 55.3563,Y 95.7786,Z 116,A 55.1536,B 24.9316,C -1.9095,E1 25.0809,E2 390.6001} C_DIS
LIN {X 57.9023,Y 94.2623,Z 116,A 53.5737,B 24.932,C -1.9052,E1 25.0847,E2 392.1852} C_DIS
LIN {X 59.9967,Y 92.9422,Z 116,A 52.3407,B 24.932,C -1.9053,E1 25.0876,E2 393.4139} C_DIS
LIN {X 62.5047,Y 91.2758,Z 116,A 50.6446,B 24.9325,C -1.8969,E1 25.0915,E2 395.1243} C_DIS
LIN {X 65.2952,Y 89.299,Z 116,A 48.9091,B 24.9327,C -1.8953,E1 25.0954,E2 396.8573} C_DIS
LIN {X 68.3499,Y 86.9837,Z 116,A 46.9201,B 24.9329,C -1.8916,E1 25.0999,E2 398.8479} C_DIS
LIN {X 70.9145,Y 84.9058,Z 116,A 45.2638,B 24.9329,C -1.8906,E1 25.1034,E2 400.5002} C_DIS
LIN {X 73.4309,Y 82.74,Z 116,A 43.3584,B 24.9338,C -1.8792,E1 25.1075,E2 402.4251} C_DIS
LIN {X 76.4536,Y 79.9551,Z 116,A 41.3341,B 24.9338,C -1.8792,E1 25.1116,E2 404.4409} C_DIS
LIN {X 78.7151,Y 77.7285,Z 116,A 39.6124,B 24.9343,C -1.8723,E1 25.115,E2 406.1716} C_DIS
LIN {X 81.4654,Y 74.8409,Z 116,A 37.7115,B 24.9341,C -1.8749,E1 25.1186,E2 408.0582} C_DIS
LIN {X 83.4668,Y 72.6025,Z 116,A 36.1044,B 24.9345,C -1.869,E1 25.1216,E2 409.6718} C_DIS
LIN {X 85.8055,Y 69.823,Z 116,A 34.2828,B 24.9346,C -1.8672,E1 25.1248,E2 411.4895} C_DIS
LIN {X 88.0407,Y 66.9856,Z 116,A 32.4947,B 24.9347,C -1.8662,E1 25.1278,E2 413.2715} C_DIS
LIN {X 90.3627,Y 63.8173,Z 116,A 30.2523,B 24.9357,C -1.852,E1 25.1315,E2 415.5365} C_DIS
LIN {X 92.7904,Y 60.2333,Z 116,A 28.294,B 24.9352,C -1.8586,E1 25.1345,E2 417.4694} C_DIS
LIN {X 93.9682,Y 58.3766,Z 116,A 26.7277,B 24.9368,C -1.8369,E1 25.1369,E2 419.0791} C_DIS
LIN {X 96.9227,Y 53.3312,Z 116,A 24.1043,B 24.9361,C -1.8464,E1 25.1405,E2 421.6664} C_DIS
LIN {X 98.8971,Y 49.572,Z 116,A 21.7434,B 24.937,C -1.8332,E1 25.1436,E2 424.0461} C_DIS
LIN {X 100.6708,Y 45.8626,Z 116,A 19.9012,B 24.9366,C -1.8398,E1 25.1457,E2 425.8626} C_DIS
LIN {X 101.6471,Y 43.6579,Z 116,A 18.3286,B 24.9378,C -1.8218,E1 25.1475,E2 427.4691} C_DIS
LIN {X 104.2077,Y 37.1326,Z 116,A 15.0141,B 24.9376,C -1.8251,E1 25.1508,E2 430.7574} C_DIS
LIN {X 105.995,Y 31.6683,Z 116,A 12.2051,B 24.9376,C -1.8236,E1 25.1532,E2 433.554} C_DIS
LIN {X 106.5898,Y 29.6095,Z 116,A 10.9031,B 24.9385,C -1.8116,E1 25.1542,E2 434.8769} C_DIS
LIN {X 107.239,Y 27.1612,Z 116,A 9.4198,B 24.9393,C -1.7999,E1 25.1553,E2 436.3792} C_DIS
LIN {X 108.0821,Y 23.5803,Z 116,A 7.6349,B 24.9393,C -1.7994,E1 25.1564,E2 438.155} C_DIS
LIN {X 108.787,Y 20.0853,Z 116,A 5.9329,B 24.9393,C -1.8,E1 25.1573,E2 439.8456} C_DIS
LIN {X 109.1719,Y 17.8719,Z 116,A 4.6512,B 24.9399,C -1.791,E1 25.1579,E2 441.1409} C_DIS
LIN {X 109.6668,Y 14.528,Z 116,A 2.8974,B 24.9403,C -1.7853,E1 25.1585,E2 442.898} C_DIS
LIN {X 110.1137,Y 10.6281,Z 116,A 0.8041,B 24.9409,C -1.7761,E1 25.1592,E2 445.0006} C_DIS
LIN {X 110.407,Y 6.9529,Z 116,A -0.9604,B 24.9409,C -1.7764,E1 25.1595,E2 446.7539} C_DIS
LIN {X 110.5724,Y 3.3956,Z 116,A -2.8259,B 24.9413,C -1.7695,E1 25.1597,E2 448.6245} C_DIS
LIN {X 110.6253,Y -0.0288,Z 116,A -4.6815,B 24.9419,C -1.7601,E1 25.1597,E2 450.4913} C_DIS
LIN {X 110.5559,Y -3.9323,Z 116,A -6.5324,B 24.9419,C -1.7612,E1 25.1597,E2 452.3287} C_DIS
LIN {X 110.4128,Y -6.867,Z 116,A -8.1112,B 24.9424,C -1.7536,E1 25.1594,E2 453.9158} C_DIS
LIN {X 110.2313,Y -9.3334,Z 116,A -9.5584,B 24.9431,C -1.742,E1 25.1591,E2 455.3819} C_DIS
LIN {X 109.7894,Y -13.5824,Z 116,A -11.5174,B 24.9429,C -1.7462,E1 25.1585,E2 457.3195} C_DIS
LIN {X 109.484,Y -15.8465,Z 116,A -12.904,B 24.9437,C -1.7332,E1 25.1579,E2 458.7284} C_DIS
LIN {X 108.8892,Y -19.5176,Z 116,A -14.722,B 24.9437,C -1.7318,E1 25.1571,E2 460.539} C_DIS
LIN {X 108.3636,Y -22.2509,Z 116,A -16.1962,B 24.9442,C -1.7257,E1 25.1563,E2 462.019} C_DIS
LIN {X 107.6082,Y -25.6631,Z 116,A -17.8782,B 24.9442,C -1.7256,E1 25.1552,E2 463.6916} C_DIS
LIN {X 106.7677,Y -28.9559,Z 116,A -20.5713,B 24.9472,C -1.6785,E1 25.1532,E2 466.4802} C_DIS
LIN {X 105.1971,Y -34.2254,Z 116,A -22.3313,B 24.9447,C -1.7179,E1 25.1518,E2 468.1373} C_DIS
LIN {X 104.4291,Y -36.5016,Z 116,A -23.7954,B 24.9456,C -1.7041,E1 25.1504,E2 469.6258} C_DIS
LIN {X 103.2325,Y -39.7645,Z 116,A -25.6852,B 24.9462,C -1.6944,E1 25.1486,E2 471.5278} C_DIS
LIN {X 102.0053,Y -42.8103,Z 116,A -27.0509,B 24.9456,C -1.7042,E1 25.1471,E2 472.8629} C_DIS
LIN {X 101.1261,Y -44.8522,Z 116,A -28.2766,B 24.946,C -1.6973,E1 25.1458,E2 474.0982} C_DIS
LIN {X 100.068,Y -47.1642,Z 116,A -30.1392,B 24.9478,C -1.669,E1 25.1435,E2 476.0176} C_DIS
LIN {X 98.4797,Y -50.3937,Z 116,A -31.5007,B 24.9467,C -1.6858,E1 25.1418,E2 477.3322} C_DIS
LIN {X 96.9562,Y -53.2694,Z 116,A -33.3341,B 24.9475,C -1.6741,E1 25.1394,E2 479.1834} C_DIS
LIN {X 95.0334,Y -56.6267,Z 116,A -35.8678,B 24.9493,C -1.6448,E1 25.1357,E2 481.7732} C_DIS
LIN {X 92.606,Y -60.5154,Z 116,A -37.3685,B 24.9473,C -1.6768,E1 25.1336,E2 483.191} C_DIS
LIN {X 90.7259,Y -63.2978,Z 116,A -39.2265,B 24.948,C -1.6666,E1 25.1306,E2 485.0639} C_DIS
LIN {X 88.6127,Y -66.2242,Z 116,A -41.2368,B 24.9487,C -1.6552,E1 25.1272,E2 487.0914} C_DIS
LIN {X 85.9306,Y -69.6686,Z 116,A -43.3681,B 24.9487,C -1.6549,E1 25.1236,E2 489.2135} C_DIS
LIN {X 83.8013,Y -72.2185,Z 116,A -45.1986,B 24.9493,C -1.6454,E1 25.1202,E2 491.0579} C_DIS
LIN {X 81.4061,Y -74.9057,Z 116,A -46.9245,B 24.9492,C -1.6468,E1 25.117,E2 492.7729} C_DIS
LIN {X 79.0814,Y -77.3576,Z 116,A -48.725,B 24.9496,C -1.6402,E1 25.1135,E2 494.5813} C_DIS
LIN {X 76.6201,Y -79.7946,Z 116,A -50.4783,B 24.9497,C -1.6376,E1 25.11,E2 496.3332} C_DIS
LIN {X 73.756,Y -82.449,Z 116,A -52.499,B 24.95,C -1.6329,E1 25.1058,E2 498.3569} C_DIS
LIN {X 70.6975,Y -85.0861,Z 116,A -54.5532,B 24.9502,C -1.6298,E1 25.1015,E2 500.4105} C_DIS
LIN {X 68.0866,Y -87.1918,Z 116,A -56.3654,B 24.9507,C -1.6227,E1 25.0975,E2 502.2328} C_DIS
LIN {X 65.3312,Y -89.2727,Z 116,A -58.0846,B 24.9507,C -1.6219,E1 25.0936,E2 503.9476} C_DIS
LIN {X 62.1901,Y -91.4889,Z 116,A -61.4357,B 24.9545,C -1.5592,E1 25.0856,E2 507.4356} C_DIS
LIN {X 55.789,Y -95.5286,Z 116,A -63.9478,B 24.9513,C -1.6124,E1 25.0799,E2 509.8142} C_DIS
LIN {X 51.3351,Y -97.9926,Z 116,A -66.5893,B 24.9516,C -1.6076,E1 25.0734,E2 512.4595} C_DIS
LIN {X 48.7416,Y -99.3087,Z 116,A -67.9868,B 24.9514,C -1.6098,E1 25.0699,E2 513.848} C_DIS
LIN {X 45.8295,Y -100.6857,Z 116,A -69.5574,B 24.9514,C -1.6114,E1 25.066,E2 515.4108} C_DIS
LIN {X 43.8331,Y -101.5707,Z 116,A -71.0128,B 24.9523,C -1.5956,E1 25.0622,E2 516.8999} C_DIS
LIN {X 39.8699,Y -103.1918,Z 116,A -73.2169,B 24.9524,C -1.5931,E1 25.0564,E2 519.1052} C_DIS
LIN {X 35.8236,Y -104.6647,Z 116,A -75.4033,B 24.9525,C -1.592,E1 25.0507,E2 521.2895} C_DIS
LIN {X 32.0647,Y -105.8774,Z 116,A -77.2729,B 24.9522,C -1.5971,E1 25.0457,E2 523.1436} C_DIS
LIN {X 28.8685,Y -106.7913,Z 116,A -78.9998,B 24.9523,C -1.5951,E1 25.0411,E2 524.8726} C_DIS
LIN {X 25.5995,Y -107.6237,Z 116,A -80.7405,B 24.9524,C -1.5935,E1 25.0364,E2 526.6143} C_DIS
LIN {X 23.5081,Y -108.0979,Z 116,A -82.0121,B 24.9529,C -1.5857,E1 25.0329,E2 527.9029} C_DIS
LIN {X 19.7348,Y -108.8501,Z 116,A -83.9249,B 24.9528,C -1.5874,E1 25.0276,E2 529.8094} C_DIS
LIN {X 16.6813,Y -109.3598,Z 116,A -85.6099,B 24.9531,C -1.5828,E1 25.023,E2 531.5037} C_DIS
LIN {X 12.947,Y -109.8643,Z 116,A -87.4893,B 24.953,C -1.5846,E1 25.0178,E2 533.3773} C_DIS
LIN {X 8.7747,Y -110.276,Z 116,A -89.6096,B 24.9529,C -1.5856,E1 25.0119,E2 535.494} C_DIS
LIN {X 5.4261,Y -110.4934,Z 116,A -91.4538,B 24.9532,C -1.5804,E1 25.0067,E2 537.3498} C_DIS
LIN {X 2.1939,Y -110.6028,Z 116,A -93.204,B 24.9534,C -1.5767,E1 25.0018,E2 539.1083} C_DIS
LIN {X 2.1939,Y -110.6028,Z 116,A -93.204,B 24.9534,C -1.5767,E1 25.0018,E2 539.1083} C_DIS
Enddeposition()
LIN {X 0.789,Y -109.7143,Z 116,A -93.464,B 24.9513,C -1.612,E1 25.0013,E2 539.2847} C_DIS
Startdeposition()
$VEL.CP = VEL_PRINT
LIN {X 4.0485,Y -109.6446,Z 116,A -91.2621,B 24.95,C -1.6335,E1 25.0076,E2 537.0323} C_DIS
LIN {X 6.7279,Y -109.5129,Z 116,A -89.989,B 24.9503,C -1.6287,E1 25.0111,E2 535.7711} C_DIS
LIN {X 9.4024,Y -109.3157,Z 116,A -88.5902,B 24.9503,C -1.6293,E1 25.015,E2 534.3715} C_DIS
LIN {X 12.1116,Y -109.0488,Z 116,A -87.1716,B 24.9503,C -1.63,E1 25.0189,E2 532.9523} C_DIS
LIN {X 14.7629,Y -108.7217,Z 116,A -85.773,B 24.9502,C -1.631,E1 25.0228,E2 531.5523} C_DIS
LIN {X 17.4201,Y -108.3276,Z 116,A -84.2252,B 24.9497,C -1.6383,E1 25.0271,E2 529.989} C_DIS
LIN {X 20.081,Y -107.8661,Z 116,A -82.8725,B 24.9497,C -1.6369,E1 25.0308,E2 528.6409} C_DIS
LIN {X 22.7306,Y -107.339,Z 116,A -81.5549,B 24.95,C -1.6342,E1 25.0344,E2 527.3314} C_DIS
LIN {X 25.352,Y -106.7503,Z 116,A -80.1543,B 24.9499,C -1.6354,E1 25.0382,E2 525.9298} C_DIS
LIN {X 28.4466,Y -105.9656,Z 116,A -78.734,B 24.9504,C -1.6266,E1 25.042,E2 524.5325} C_DIS
LIN {X 30.564,Y -105.3764,Z 116,A -77.3543,B 24.9497,C -1.6378,E1 25.0458,E2 523.1287} C_DIS
LIN {X 33.1213,Y -104.6007,Z 116,A -75.96,B 24.9497,C -1.6394,E1 25.0495,E2 521.7331} C_DIS
LIN {X 35.8143,Y -103.7089,Z 116,A -74.5338,B 24.9497,C -1.6389,E1 25.0533,E2 520.3108} C_DIS
LIN {X 38.2566,Y -102.8335,Z 116,A -73.1401,B 24.9495,C -1.6424,E1 25.0569,E2 518.9118} C_DIS
LIN {X 40.7629,Y -101.8661,Z 116,A -71.7413,B 24.9493,C -1.6442,E1 25.0606,E2 517.5119} C_DIS
LIN {X 43.245,Y -100.8374,Z 116,A -70.3354,B 24.9493,C -1.6464,E1 25.0642,E2 516.1041} C_DIS
LIN {X 45.7013,Y -99.7483,Z 116,A -68.9415,B 24.9491,C -1.6481,E1 25.0677,E2 514.7095} C_DIS
LIN {X 48.1166,Y -98.6059,Z 116,A -67.5454,B 24.949,C -1.6504,E1 25.0713,E2 513.3116} C_DIS
LIN {X 50.5164,Y -97.3983,Z 116,A -66.1353,B 24.9488,C -1.6531,E1 25.0748,E2 511.8991} C_DIS
LIN {X 52.9166,Y -96.1154,Z 116,A -64.5675,B 24.9482,C -1.662,E1 25.0787,E2 510.3148} C_DIS
LIN {X 55.2514,Y -94.7925,Z 116,A -63.3376,B 24.9485,C -1.6571,E1 25.0816,E2 509.1002} C_DIS
LIN {X 57.5266,Y -93.4291,Z 116,A -61.9564,B 24.9484,C -1.6595,E1 25.0849,E2 507.7176} C_DIS
LIN {X 59.7864,Y -91.9992,Z 116,A -60.5662,B 24.9482,C -1.662,E1 25.0882,E2 506.3262} C_DIS
LIN {X 62.0693,Y -90.4751,Z 116,A -58.9764,B 24.9476,C -1.6717,E1 25.0919,E2 504.7186} C_DIS
LIN {X 65.3822,Y -88.1106,Z 116,A -57.0313,B 24.9478,C -1.6682,E1 25.0962,E2 502.7886} C_DIS
LIN {X 67.5137,Y -86.4883,Z 116,A -55.631,B 24.9477,C -1.6713,E1 25.0993,E2 501.3862} C_DIS
LIN {X 69.6062,Y -84.8135,Z 116,A -54.2375,B 24.9475,C -1.6742,E1 25.1024,E2 499.9912} C_DIS
LIN {X 72.1058,Y -82.6962,Z 116,A -52.5116,B 24.9472,C -1.6788,E1 25.106,E2 498.2612} C_DIS
LIN {X 74.3837,Y -80.6538,Z 116,A -50.8965,B 24.9469,C -1.6833,E1 25.1094,E2 496.6418} C_DIS
LIN {X 76.628,Y -78.527,Z 116,A -49.3366,B 24.9469,C -1.6848,E1 25.1125,E2 495.085} C_DIS
LIN {X 78.5285,Y -76.6265,Z 116,A -47.941,B 24.9466,C -1.6879,E1 25.1153,E2 493.688} C_DIS
LIN {X 80.7177,Y -74.314,Z 116,A -46.2382,B 24.9462,C -1.6939,E1 25.1185,E2 491.9784} C_DIS
LIN {X 82.7562,Y -72.0371,Z 116,A -44.634,B 24.9459,C -1.6984,E1 25.1215,E2 490.3708} C_DIS
LIN {X 84.8149,Y -69.6044,Z 116,A -43.0443,B 24.9459,C -1.6995,E1 25.1243,E2 488.7859} C_DIS
LIN {X 86.499,Y -67.5001,Z 116,A -41.649,B 24.9457,C -1.7027,E1 25.1267,E2 487.3895} C_DIS
LIN {X 88.4233,Y -64.9557,Z 116,A -39.9617,B 24.9453,C -1.7083,E1 25.1296,E2 485.6972} C_DIS
LIN {X 90.4847,Y -62.0552,Z 116,A -38.1522,B 24.9451,C -1.7112,E1 25.1325,E2 483.8895} C_DIS
LIN {X 92.0037,Y -59.7795,Z 116,A -36.7292,B 24.9449,C -1.715,E1 25.1346,E2 482.4647} C_DIS
LIN {X 93.4238,Y -57.5352,Z 116,A -35.3498,B 24.9446,C -1.7187,E1 25.1367,E2 481.0836} C_DIS
LIN {X 94.8058,Y -55.2283,Z 116,A -33.9541,B 24.9444,C -1.7224,E1 25.1387,E2 479.6864} C_DIS
LIN {X 96.7616,Y -51.7256,Z 116,A -31.8681,B 24.944,C -1.7282,E1 25.1415,E2 477.5976} C_DIS
LIN {X 97.9924,Y -49.3539,Z 116,A -30.4817,B 24.9438,C -1.732,E1 25.1432,E2 476.2096} C_DIS
LIN {X 99.1607,Y -46.962,Z 116,A -29.002,B 24.9432,C -1.7402,E1 25.145,E2 474.7184} C_DIS
LIN {X 100.3064,Y -44.4631,Z 116,A -27.6688,B 24.9432,C -1.74,E1 25.1466,E2 473.393} C_DIS
LIN {X 101.3653,Y -41.993,Z 116,A -26.2771,B 24.943,C -1.7438,E1 25.1481,E2 472} C_DIS
LIN {X 102.3633,Y -39.4978,Z 116,A -24.8857,B 24.9428,C -1.7476,E1 25.1495,E2 470.6074} C_DIS
LIN {X 103.4224,Y -36.6307,Z 116,A -23.4672,B 24.943,C -1.7447,E1 25.1508,E2 469.2037} C_DIS
LIN {X 104.2908,Y -34.0796,Z 116,A -22.0701,B 24.9427,C -1.7486,E1 25.1521,E2 467.8051} C_DIS
LIN {X 104.9618,Y -31.9568,Z 116,A -20.7501,B 24.942,C -1.7594,E1 25.1532,E2 466.4674} C_DIS
LIN {X 105.7616,Y -29.202,Z 116,A -19.2885,B 24.9418,C -1.7625,E1 25.1543,E2 465.0067} C_DIS
LIN {X 106.4351,Y -26.6439,Z 116,A -17.8963,B 24.9415,C -1.7674,E1 25.1553,E2 463.611} C_DIS
LIN {X 107.0914,Y -23.8656,Z 116,A -16.3799,B 24.9411,C -1.7734,E1 25.1562,E2 462.0893} C_DIS
LIN {X 107.6142,Y -21.3894,Z 116,A -15.0922,B 24.9409,C -1.7761,E1 25.1569,E2 460.8027} C_DIS
LIN {X 108.1082,Y -18.7331,Z 116,A -13.7028,B 24.9406,C -1.7797,E1 25.1576,E2 459.4129} C_DIS
LIN {X 108.5346,Y -16.0801,Z 116,A -12.3094,B 24.9404,C -1.7838,E1 25.1582,E2 458.018} C_DIS
LIN {X 108.9067,Y -13.3244,Z 116,A -10.904,B 24.9402,C -1.7864,E1 25.1587,E2 456.6147} C_DIS
LIN {X 109.1903,Y -10.7614,Z 116,A -9.5193,B 24.9398,C -1.7925,E1 25.1591,E2 455.2239} C_DIS
LIN {X 109.4231,Y -8.0577,Z 116,A -8.1094,B 24.9395,C -1.7968,E1 25.1594,E2 453.8122} C_DIS
LIN {X 109.5875,Y -5.3782,Z 116,A -6.7171,B 24.9392,C -1.801,E1 25.1596,E2 452.4184} C_DIS
LIN {X 109.6863,Y -2.6953,Z 116,A -5.2723,B 24.9388,C -1.8075,E1 25.1598,E2 450.9669} C_DIS
LIN {X 109.7183,Y -0.0103,Z 116,A -3.9787,B 24.9388,C -1.8071,E1 25.1598,E2 449.6817} C_DIS
LIN {X 109.6867,Y 2.673,Z 116,A -2.5339,B 24.9383,C -1.8136,E1 25.1598,E2 448.2302} C_DIS
LIN {X 109.5869,Y 5.39,Z 116,A -1.1311,B 24.9381,C -1.8175,E1 25.1595,E2 446.8267} C_DIS
LIN {X 109.4223,Y 8.0686,Z 116,A 0.2592,B 24.9378,C -1.8215,E1 25.1593,E2 445.4352} C_DIS
LIN {X 109.1922,Y 10.7421,Z 116,A 1.656,B 24.9375,C -1.8258,E1 25.1589,E2 444.0365} C_DIS
LIN {X 108.8924,Y 13.4453,Z 116,A 3.0551,B 24.9373,C -1.8294,E1 25.1585,E2 442.6372} C_DIS
LIN {X 108.5287,Y 16.1199,Z 116,A 4.4494,B 24.937,C -1.8332,E1 25.1579,E2 441.2421} C_DIS
LIN {X 108.104,Y 18.7585,Z 116,A 5.8499,B 24.9367,C -1.8378,E1 25.1573,E2 439.8389} C_DIS
LIN {X 107.535,Y 21.7763,Z 116,A 7.4571,B 24.9363,C -1.8431,E1 25.1564,E2 438.2287} C_DIS
LIN {X 106.9151,Y 24.6386,Z 116,A 8.8515,B 24.9364,C -1.8418,E1 25.1556,E2 436.8454} C_DIS
LIN {X 106.0948,Y 27.9685,Z 116,A 10.7831,B 24.9356,C -1.8536,E1 25.1542,E2 434.8972} C_DIS
LIN {X 105.3736,Y 30.5734,Z 116,A 12.209,B 24.9352,C -1.8586,E1 25.1531,E2 433.4676} C_DIS
LIN {X 104.5914,Y 33.1507,Z 116,A 13.537,B 24.9352,C -1.8594,E1 25.152,E2 432.1454} C_DIS
LIN {X 103.6794,Y 35.8982,Z 116,A 14.9341,B 24.9352,C -1.8588,E1 25.1508,E2 430.7575} C_DIS
LIN {X 102.8486,Y 38.2166,Z 116,A 16.3146,B 24.9347,C -1.8669,E1 25.1495,E2 429.3657} C_DIS
LIN {X 101.8892,Y 40.7049,Z 116,A 17.7021,B 24.9344,C -1.8707,E1 25.148,E2 427.9768} C_DIS
LIN {X 100.8373,Y 43.2454,Z 116,A 19.124,B 24.9341,C -1.8743,E1 25.1465,E2 426.5543} C_DIS
LIN {X 99.7481,Y 45.7017,Z 116,A 20.514,B 24.9339,C -1.8777,E1 25.1449,E2 425.1637} C_DIS
LIN {X 98.519,Y 48.2923,Z 116,A 22.0516,B 24.9335,C -1.8838,E1 25.143,E2 423.6201} C_DIS
LIN {X 96.7616,Y 51.7257,Z 116,A 24.0186,B 24.9332,C -1.8873,E1 25.1405,E2 421.6552} C_DIS
LIN {X 95.4607,Y 54.0888,Z 116,A 25.4283,B 24.933,C -1.8912,E1 25.1386,E2 420.2437} C_DIS
LIN {X 94.1094,Y 56.4072,Z 116,A 26.8063,B 24.9328,C -1.8939,E1 25.1366,E2 418.8663} C_DIS
LIN {X 92.696,Y 58.7009,Z 116,A 28.209,B 24.9325,C -1.8975,E1 25.1345,E2 417.4623} C_DIS
LIN {X 91.2307,Y 60.9533,Z 116,A 29.5986,B 24.9323,C -1.9005,E1 25.1324,E2 416.0724} C_DIS
LIN {X 89.7021,Y 63.1813,Z 116,A 31.1809,B 24.9315,C -1.9117,E1 25.1298,E2 414.4716} C_DIS
LIN {X 88.0158,Y 65.5084,Z 116,A 32.5614,B 24.9316,C -1.9101,E1 25.1276,E2 413.1014} C_DIS
LIN {X 86.074,Y 68.038,Z 116,A 34.1524,B 24.9316,C -1.9109,E1 25.1248,E2 411.516} C_DIS
LIN {X 84.3812,Y 70.1264,Z 116,A 35.5473,B 24.9313,C -1.9139,E1 25.1224,E2 410.1205} C_DIS
LIN {X 82.6327,Y 72.1785,Z 116,A 36.9483,B 24.9311,C -1.9168,E1 25.1198,E2 408.7189} C_DIS
LIN {X 80.8444,Y 74.176,Z 116,A 38.3414,B 24.9309,C -1.9197,E1 25.1172,E2 407.3252} C_DIS
LIN {X 78.7662,Y 76.3799,Z 116,A 39.9535,B 24.9306,C -1.9245,E1 25.1141,E2 405.7087} C_DIS
LIN {X 76.1436,Y 78.994,Z 116,A 41.8404,B 24.9304,C -1.9266,E1 25.1103,E2 403.8248} C_DIS
LIN {X 74.1824,Y 80.8385,Z 116,A 43.2453,B 24.9302,C -1.9295,E1 25.1074,E2 402.4189} C_DIS
LIN {X 72.1657,Y 82.6438,Z 116,A 44.6995,B 24.9299,C -1.9341,E1 25.1044,E2 400.9596} C_DIS
LIN {X 69.6087,Y 84.8114,Z 116,A 46.3919,B 24.9299,C -1.9349,E1 25.1008,E2 399.2718} C_DIS
LIN {X 67.5048,Y 86.4953,Z 116,A 47.7934,B 24.9296,C -1.9372,E1 25.0977,E2 397.8698} C_DIS
LIN {X 65.0194,Y 88.3767,Z 116,A 49.2742,B 24.9299,C -1.9338,E1 25.0944,E2 396.4025} C_DIS
LIN {X 62.9183,Y 89.885,Z 116,A 50.6265,B 24.9297,C -1.9362,E1 25.0913,E2 395.0493} C_DIS
LIN {X 60.9509,Y 91.2322,Z 116,A 52.0074,B 24.9291,C -1.9441,E1 25.0881,E2 393.6544} C_DIS
LIN {X 58.6858,Y 92.7055,Z 116,A 53.5407,B 24.9286,C -1.9516,E1 25.0845,E2 392.1084} C_DIS
LIN {X 56.4109,Y 94.1071,Z 116,A 54.8023,B 24.9289,C -1.9479,E1 25.0815,E2 390.8593} C_DIS
LIN {X 54.0407,Y 95.4877,Z 116,A 56.208,B 24.9288,C -1.9489,E1 25.0781,E2 389.4557} C_DIS
LIN {X 51.7276,Y 96.7605,Z 116,A 57.7419,B 24.9282,C -1.9574,E1 25.0743,E2 387.9059} C_DIS
LIN {X 49.3179,Y 98.0106,Z 116,A 59.0206,B 24.9285,C -1.9533,E1 25.0711,E2 386.6405} C_DIS
LIN {X 46.9031,Y 99.1889,Z 116,A 60.4132,B 24.9284,C -1.9546,E1 25.0676,E2 385.2485} C_DIS
LIN {X 44.4603,Y 100.3077,Z 116,A 61.8196,B 24.9282,C -1.9563,E1 25.0641,E2 383.8414} C_DIS
LIN {X 41.5324,Y 101.5529,Z 116,A 63.2449,B 24.9288,C -1.9482,E1 25.0604,E2 382.4388} C_DIS
LIN {X 39.496,Y 102.3641,Z 116,A 64.6153,B 24.9281,C -1.9588,E1 25.0568,E2 381.0463} C_DIS
LIN {X 36.9641,Y 103.3054,Z 116,A 66.0221,B 24.928,C -1.9599,E1 25.0531,E2 379.6397} C_DIS
LIN {X 34.396,Y 104.1885,Z 116,A 67.5507,B 24.9275,C -1.9658,E1 25.0491,E2 378.1001} C_DIS
LIN {X 31.8622,Y 104.9911,Z 116,A 68.968,B 24.9274,C -1.9681,E1 25.0453,E2 376.68} C_DIS
LIN {X 29.2829,Y 105.7395,Z 116,A 70.3708,B 24.9274,C -1.969,E1 25.0415,E2 375.2772} C_DIS
LIN {X 26.6428,Y 106.4354,Z 116,A 71.639,B 24.9277,C -1.9633,E1 25.0381,E2 374.0245} C_DIS
LIN {X 22.7147,Y 107.3423,Z 116,A 73.7493,B 24.9277,C -1.9646,E1 25.0324,E2 371.914} C_DIS
LIN {X 20.0607,Y 107.8698,Z 116,A 75.161,B 24.9276,C -1.9652,E1 25.0285,E2 370.5026} C_DIS
LIN {X 17.4274,Y 108.3265,Z 116,A 76.563,B 24.9276,C -1.9659,E1 25.0246,E2 369.1004} C_DIS
LIN {X 14.7688,Y 108.7209,Z 116,A 77.9996,B 24.9274,C -1.9676,E1 25.0206,E2 367.6609} C_DIS
LIN {X 12.077,Y 109.0526,Z 116,A 79.3675,B 24.9275,C -1.9659,E1 25.0169,E2 366.2981} C_DIS
LIN {X 9.4037,Y 109.3156,Z 116,A 80.9532,B 24.927,C -1.9736,E1 25.0124,E2 364.695} C_DIS
LIN {X 6.7089,Y 109.514,Z 116,A 82.1799,B 24.9275,C -1.966,E1 25.009,E2 363.4869} C_DIS
LIN {X 4.0275,Y 109.6454,Z 116,A 83.7414,B 24.9271,C -1.9725,E1 25.0046,E2 361.9105} C_DIS
LIN {X 1.359,Y 109.7109,Z 116,A 84.9855,B 24.9275,C -1.9661,E1 25.0012,E2 360.6817} C_DIS
LIN {X -1.3393,Y 109.7112,Z 116,A 86.3953,B 24.9275,C -1.9658,E1 24.9973,E2 359.2725} C_DIS
LIN {X -4.0574,Y 109.6442,Z 116,A 87.8071,B 24.9275,C -1.9651,E1 24.9933,E2 357.8622} C_DIS
LIN {X -6.74,Y 109.5121,Z 116,A 89.2141,B 24.9276,C -1.9648,E1 24.9894,E2 356.4557} C_DIS
LIN {X -9.4183,Y 109.3144,Z 116,A 90.6213,B 24.9276,C -1.9643,E1 24.9855,E2 355.0488} C_DIS
LIN {X -12.0904,Y 109.0512,Z 116,A 92.0274,B 24.9277,C -1.9637,E1 24.9816,E2 353.6434} C_DIS
LIN {X -15.2945,Y 108.6462,Z 116,A 93.4753,B 24.9285,C -1.9531,E1 24.9777,E2 352.2196} C_DIS
LIN {X -17.4297,Y 108.3262,Z 116,A 94.8454,B 24.9278,C -1.962,E1 24.9738,E2 350.8271} C_DIS
LIN {X -20.0925,Y 107.8639,Z 116,A 96.2546,B 24.9279,C -1.9609,E1 24.9699,E2 349.4192} C_DIS
LIN {X -22.7135,Y 107.3426,Z 116,A 97.8397,B 24.9274,C -1.9673,E1 24.9656,E2 347.8169} C_DIS
LIN {X -26.6791,Y 106.4263,Z 116,A 99.7784,B 24.9281,C -1.9578,E1 24.9603,E2 345.8982} C_DIS
LIN {X -29.3424,Y 105.7226,Z 116,A 101.2152,B 24.9282,C -1.9563,E1 24.9565,E2 344.4628} C_DIS
LIN {X -31.9424,Y 104.9662,Z 116,A 102.6,B 24.9285,C -1.9535,E1 24.9528,E2 343.0822} C_DIS
LIN {X -34.3453,Y 104.2049,Z 116,A 103.964,B 24.9285,C -1.9539,E1 24.9492,E2 341.7149} C_DIS
LIN {X -37.3812,Y 103.1533,Z 116,A 105.445,B 24.9292,C -1.944,E1 24.9453,E2 340.2546} C_DIS
LIN {X -39.4782,Y 102.3709,Z 116,A 106.8205,B 24.9287,C -1.9506,E1 24.9417,E2 338.8605} C_DIS
LIN {X -41.9639,Y 101.3772,Z 116,A 108.2228,B 24.9287,C -1.9488,E1 24.938,E2 337.4594} C_DIS
LIN {X -44.4349,Y 100.3187,Z 116,A 109.6383,B 24.9289,C -1.9472,E1 24.9344,E2 336.0443} C_DIS
LIN {X -47.3611,Y 98.9689,Z 116,A 111.0811,B 24.9298,C -1.9351,E1 24.9308,E2 334.6265} C_DIS
LIN {X -49.3286,Y 98.0053,Z 116,A 112.4676,B 24.9292,C -1.9428,E1 24.9273,E2 333.2181} C_DIS
LIN {X -51.7961,Y 96.7233,Z 116,A 113.8898,B 24.9295,C -1.9392,E1 24.9238,E2 331.8006} C_DIS
LIN {X -54.0861,Y 95.4622,Z 116,A 115.3009,B 24.9295,C -1.9386,E1 24.9204,E2 330.3869} C_DIS
LIN {X -56.4186,Y 94.1024,Z 116,A 116.7045,B 24.9297,C -1.9358,E1 24.917,E2 328.9857} C_DIS
LIN {X -58.6916,Y 92.7018,Z 116,A 118.1118,B 24.9299,C -1.9337,E1 24.9137,E2 327.579} C_DIS
LIN {X -60.9419,Y 91.2382,Z 116,A 119.5187,B 24.9301,C -1.9311,E1 24.9104,E2 326.1735} C_DIS
LIN {X -63.17,Y 89.71,Z 116,A 120.9817,B 24.9301,C -1.9303,E1 24.907,E2 324.7074} C_DIS
LIN {X -65.3721,Y 88.1182,Z 116,A 122.3537,B 24.9305,C -1.9255,E1 24.9039,E2 323.342} C_DIS
LIN {X -67.4916,Y 86.5056,Z 116,A 123.7582,B 24.9307,C -1.9231,E1 24.9008,E2 321.9381} C_DIS
LIN {X -69.569,Y 84.8436,Z 116,A 125.1541,B 24.9309,C -1.9203,E1 24.8978,E2 320.5436} C_DIS
LIN {X -71.6044,Y 83.1328,Z 116,A 126.7463,B 24.9305,C -1.9251,E1 24.8944,E2 318.9339} C_DIS
LIN {X -74.6569,Y 80.4032,Z 116,A 128.895,B 24.9309,C -1.9205,E1 24.89,E2 316.7874} C_DIS
LIN {X -77.5251,Y 77.6409,Z 116,A 130.7865,B 24.9317,C -1.9082,E1 24.8862,E2 314.9173} C_DIS
LIN {X -79.5498,Y 75.5647,Z 116,A 132.2931,B 24.932,C -1.9042,E1 24.8833,E2 313.4138} C_DIS
LIN {X -81.3249,Y 73.6515,Z 116,A 133.7822,B 24.932,C -1.9056,E1 24.8805,E2 311.9147} C_DIS
LIN {X -83.5054,Y 71.1671,Z 116,A 135.4116,B 24.9325,C -1.8974,E1 24.8776,E2 310.2974} C_DIS
LIN {X -85.5871,Y 68.6517,Z 116,A 137.3043,B 24.9323,C -1.9001,E1 24.8742,E2 308.3894} C_DIS
LIN {X -87.9908,Y 65.5417,Z 116,A 139.217,B 24.9331,C -1.8892,E1 24.871,E2 306.4936} C_DIS
LIN {X -89.7136,Y 63.1649,Z 116,A 140.7368,B 24.9334,C -1.8845,E1 24.8685,E2 304.9778} C_DIS
LIN {X -91.2205,Y 60.9685,Z 116,A 142.1397,B 24.9337,C -1.881,E1 24.8663,E2 303.576} C_DIS
LIN {X -92.6887,Y 58.7123,Z 116,A 143.554,B 24.9339,C -1.8774,E1 24.8642,E2 302.1634} C_DIS
LIN {X -94.0845,Y 56.4482,Z 116,A 145.0753,B 24.9339,C -1.8784,E1 24.862,E2 300.6316} C_DIS
LIN {X -95.4732,Y 54.0666,Z 116,A 146.3991,B 24.9345,C -1.8698,E1 24.8602,E2 299.3214} C_DIS
LIN {X -96.7685,Y 51.7127,Z 116,A 147.811,B 24.9347,C -1.866,E1 24.8583,E2 297.9112} C_DIS
LIN {X -98.0056,Y 49.328,Z 116,A 149.3722,B 24.9346,C -1.8679,E1 24.8563,E2 296.3372} C_DIS
LIN {X -99.7689,Y 45.656,Z 116,A 151.349,B 24.9354,C -1.8557,E1 24.854,E2 294.3787} C_DIS
LIN {X -100.9133,Y 43.0656,Z 116,A 152.7807,B 24.9359,C -1.8494,E1 24.8524,E2 292.954} C_DIS
LIN {X -101.8863,Y 40.7123,Z 116,A 154.1843,B 24.9359,C -1.8481,E1 24.8509,E2 291.5457} C_DIS
LIN {X -102.9519,Y 37.9333,Z 116,A 155.6189,B 24.9366,C -1.8388,E1 24.8495,E2 290.1253} C_DIS
LIN {X -103.7514,Y 35.6931,Z 116,A 157.014,B 24.9365,C -1.8407,E1 24.8482,E2 288.7178} C_DIS
LIN {X -104.5982,Y 33.1293,Z 116,A 158.4298,B 24.9368,C -1.8365,E1 24.847,E2 287.304} C_DIS
LIN {X -105.3829,Y 30.5413,Z 116,A 159.8474,B 24.9371,C -1.8322,E1 24.8459,E2 285.8883} C_DIS
LIN {X -106.0938,Y 27.9721,Z 116,A 161.2701,B 24.9373,C -1.8289,E1 24.8448,E2 284.4651} C_DIS
LIN {X -106.7534,Y 25.3386,Z 116,A 162.8367,B 24.9373,C -1.83,E1 24.8438,E2 282.8868} C_DIS
LIN {X -107.3419,Y 22.7167,Z 116,A 164.0893,B 24.9379,C -1.8198,E1 24.8431,E2 281.6512} C_DIS
LIN {X -107.8631,Y 20.097,Z 116,A 165.4973,B 24.9382,C -1.8158,E1 24.8423,E2 280.2443} C_DIS
LIN {X -108.3172,Y 17.4834,Z 116,A 166.8926,B 24.9385,C -1.8117,E1 24.8417,E2 278.8505} C_DIS
LIN {X -108.7207,Y 14.77,Z 116,A 168.5007,B 24.9383,C -1.8137,E1 24.841,E2 277.228} C_DIS
LIN {X -109.1923,Y 10.7414,Z 116,A 170.474,B 24.9392,C -1.8014,E1 24.8405,E2 275.2724} C_DIS
LIN {X -109.4226,Y 8.0639,Z 116,A 171.8874,B 24.9395,C -1.7972,E1 24.8401,E2 273.8605} C_DIS
LIN {X -109.5874,Y 5.3812,Z 116,A 173.3004,B 24.9397,C -1.793,E1 24.8399,E2 272.449} C_DIS
LIN {X -109.6931,Y 2.3249,Z 116,A 174.9453,B 24.94,C -1.7896,E1 24.8399,E2 270.8022} C_DIS
LIN {X -109.7107,Y -1.37,Z 116,A 176.8384,B 24.9405,C -1.782,E1 24.8399,E2 268.9159} C_DIS
LIN {X -109.6443,Y -4.0572,Z 116,A 178.2518,B 24.9408,C -1.7778,E1 24.8399,E2 267.5039} C_DIS
LIN {X -109.512,Y -6.742,Z 116,A 179.6672,B 24.941,C -1.7737,E1 24.8402,E2 266.0898} C_DIS
LIN {X -109.264,Y -9.9645,Z 116,A -178.6061,B 24.9413,C -1.7698,E1 24.8406,E2 264.362} C_DIS
LIN {X -108.8914,Y -13.4532,Z 116,A -176.7897,B 24.9417,C -1.7633,E1 24.8411,E2 262.5502} C_DIS
LIN {X -108.5292,Y -16.1163,Z 116,A -175.3768,B 24.942,C -1.7592,E1 24.8417,E2 261.1388} C_DIS
LIN {X -108.1046,Y -18.755,Z 116,A -173.9585,B 24.9422,C -1.7557,E1 24.8423,E2 259.7205} C_DIS
LIN {X -107.4996,Y -21.9486,Z 116,A -172.4332,B 24.943,C -1.7438,E1 24.8431,E2 258.2144} C_DIS
LIN {X -107.0446,Y -24.0778,Z 116,A -171.1208,B 24.9428,C -1.7469,E1 24.8439,E2 256.8869} C_DIS
LIN {X -106.4259,Y -26.6807,Z 116,A -169.7133,B 24.9431,C -1.743,E1 24.8449,E2 255.4806} C_DIS
LIN {X -105.7476,Y -29.2538,Z 116,A -168.2931,B 24.9433,C -1.7399,E1 24.8459,E2 254.0595} C_DIS
LIN {X -104.9937,Y -31.8537,Z 116,A -166.8825,B 24.9436,C -1.7354,E1 24.847,E2 252.6513} C_DIS
LIN {X -104.1779,Y -34.4282,Z 116,A -165.4233,B 24.9437,C -1.7331,E1 24.8483,E2 251.1895} C_DIS
LIN {X -103.3092,Y -36.9534,Z 116,A -164.0485,B 24.944,C -1.7281,E1 24.8496,E2 249.8185} C_DIS
LIN {X -102.1552,Y -40.0278,Z 116,A -162.5913,B 24.945,C -1.7132,E1 24.851,E2 248.3887} C_DIS
LIN {X -101.3656,Y -41.9923,Z 116,A -161.2136,B 24.9445,C -1.7204,E1 24.8524,E2 246.9862} C_DIS
LIN {X -100.3005,Y -44.4763,Z 116,A -159.8,B 24.9448,C -1.7164,E1 24.854,E2 245.5744} C_DIS
LIN {X -99.1875,Y -46.9061,Z 116,A -158.2375,B 24.9446,C -1.7189,E1 24.8559,E2 243.9975} C_DIS
LIN {X -97.998,Y -49.343,Z 116,A -156.9716,B 24.9453,C -1.7091,E1 24.8574,E2 242.7481} C_DIS
LIN {X -96.7617,Y -51.7254,Z 116,A -155.5616,B 24.9455,C -1.7055,E1 24.8593,E2 241.3391} C_DIS
LIN {X -95.4673,Y -54.0771,Z 116,A -153.9768,B 24.9453,C -1.7088,E1 24.8615,E2 239.7381} C_DIS
LIN {X -94.0991,Y -56.4242,Z 116,A -152.731,B 24.9459,C -1.6983,E1 24.8632,E2 238.5109} C_DIS
LIN {X -92.6969,Y -58.6995,Z 116,A -151.3128,B 24.9461,C -1.6955,E1 24.8653,E2 237.0922} C_DIS
LIN {X -91.2313,Y -60.9523,Z 116,A -149.799,B 24.9461,C -1.6962,E1 24.8677,E2 235.5692} C_DIS
LIN {X -89.696,Y -63.1899,Z 116,A -148.4899,B 24.9466,C -1.6884,E1 24.8697,E2 234.2722} C_DIS
LIN {X -88.1428,Y -65.3388,Z 116,A -147.0909,B 24.9468,C -1.6855,E1 24.872,E2 232.8734} C_DIS
LIN {X -86.1373,Y -67.9578,Z 116,A -145.2344,B 24.9467,C -1.6866,E1 24.8752,E2 231.0055} C_DIS
LIN {X -83.9529,Y -70.6417,Z 116,A -143.5422,B 24.9472,C -1.6778,E1 24.8782,E2 229.3264} C_DIS
LIN {X -82.0702,Y -72.8191,Z 116,A -142.1164,B 24.9477,C -1.6713,E1 24.8808,E2 227.9095} C_DIS
LIN {X -80.378,Y -74.684,Z 116,A -140.5308,B 24.9472,C -1.679,E1 24.8839,E2 226.2986} C_DIS
LIN {X -78.0584,Y -77.1024,Z 116,A -138.9508,B 24.9478,C -1.6685,E1 24.8869,E2 224.7368} C_DIS
LIN {X -75.9279,Y -79.2019,Z 116,A -137.3382,B 24.9479,C -1.6672,E1 24.8902,E2 223.1205} C_DIS
LIN {X -73.2729,Y -81.6639,Z 116,A -135.45,B 24.9482,C -1.6633,E1 24.8941,E2 221.2341} C_DIS
LIN {X -71.1492,Y -83.5206,Z 116,A -134.0048,B 24.9484,C -1.6593,E1 24.8971,E2 219.7926} C_DIS
LIN {X -69.0871,Y -85.2342,Z 116,A -132.5989,B 24.9486,C -1.6569,E1 24.9001,E2 218.3872} C_DIS
LIN {X -66.7112,Y -87.1069,Z 116,A -130.9733,B 24.9486,C -1.6559,E1 24.9037,E2 216.7581} C_DIS
LIN {X -64.2667,Y -88.9277,Z 116,A -129.4085,B 24.9489,C -1.652,E1 24.9072,E2 215.197} C_DIS
LIN {X -62.0567,Y -90.4837,Z 116,A -128.0063,B 24.949,C -1.6493,E1 24.9105,E2 213.7964} C_DIS
LIN {X -59.685,Y -92.0643,Z 116,A -126.5825,B 24.9493,C -1.6444,E1 24.9138,E2 212.3798} C_DIS
LIN {X -57.5511,Y -93.4142,Z 116,A -125.185,B 24.9493,C -1.6455,E1 24.9171,E2 210.9751} C_DIS
LIN {X -55.2419,Y -94.7981,Z 116,A -123.7745,B 24.9493,C -1.6436,E1 24.9205,E2 209.5648} C_DIS
LIN {X -51.7082,Y -96.7708,Z 116,A -121.4916,B 24.9491,C -1.6476,E1 24.9261,E2 207.266} C_DIS
LIN {X -49.3108,Y -98.0141,Z 116,A -120.2384,B 24.9496,C -1.6394,E1 24.9292,E2 206.0288} C_DIS
LIN {X -46.9093,Y -99.186,Z 116,A -118.839,B 24.9497,C -1.6379,E1 24.9327,E2 204.6293} C_DIS
LIN {X -44.3379,Y -100.361,Z 116,A -117.4188,B 24.95,C -1.634,E1 24.9363,E2 203.215} C_DIS
LIN {X -41.9964,Y -101.3639,Z 116,A -116.0237,B 24.9499,C -1.6352,E1 24.9399,E2 201.8138} C_DIS
LIN {X -39.5018,Y -102.3618,Z 116,A -114.6054,B 24.9499,C -1.6345,E1 24.9436,E2 200.3942} C_DIS
LIN {X -36.9456,Y -103.3119,Z 116,A -113.2011,B 24.9501,C -1.6324,E1 24.9473,E2 198.992} C_DIS
LIN {X -34.4183,Y -104.1812,Z 116,A -111.7937,B 24.9501,C -1.6318,E1 24.951,E2 197.5836} C_DIS
LIN {X -31.8484,Y -104.9954,Z 116,A -110.3765,B 24.9501,C -1.6311,E1 24.9548,E2 196.1654} C_DIS
LIN {X -29.2493,Y -105.7488,Z 116,A -108.9758,B 24.9502,C -1.6297,E1 24.9586,E2 194.7659} C_DIS
LIN {X -26.5556,Y -106.4566,Z 116,A -107.5636,B 24.9504,C -1.6271,E1 24.9624,E2 193.3578} C_DIS
LIN {X -24.0174,Y -107.0583,Z 116,A -106.1502,B 24.9504,C -1.6285,E1 24.9662,E2 191.9392} C_DIS
LIN {X -21.4031,Y -107.6116,Z 116,A -104.7463,B 24.9504,C -1.6283,E1 24.9701,E2 190.5342} C_DIS
LIN {X -18.7463,Y -108.106,Z 116,A -103.1523,B 24.9499,C -1.6354,E1 24.9745,E2 188.9218} C_DIS
LIN {X -14.7652,Y -108.7214,Z 116,A -101.2351,B 24.9504,C -1.6271,E1 24.9798,E2 187.0226} C_DIS
LIN {X -12.0853,Y -109.0517,Z 116,A -99.8236,B 24.9504,C -1.6269,E1 24.9837,E2 185.6105} C_DIS
LIN {X -9.3943,Y -109.3164,Z 116,A -98.3322,B 24.9502,C -1.6302,E1 24.9878,E2 184.1107} C_DIS
LIN {X -5.3957,Y -109.5866,Z 116,A -96.3191,B 24.9504,C -1.6269,E1 24.9934,E2 182.1047} C_DIS
LIN {X -2.7165,Y -109.6856,Z 116,A -94.9197,B 24.9504,C -1.6271,E1 24.9973,E2 180.7047} C_DIS
LIN {X -0.0176,Y -109.7193,Z 116,A -93.5013,B 24.9504,C -1.6277,E1 25.0013,E2 179.2847} C_DIS
LIN {X -0.0176,Y -109.7193,Z 116,A -93.5013,B 24.9504,C -1.6277,E1 25.0013,E2 179.2847} C_DIS
Enddeposition()
LIN {X 0.8116,Y -115.8194,Z 117,A -93.2512,B 24.9566,C -1.5217,E1 25.0013,E2 179.286} C_DIS
Startdeposition()
$VEL.CP = VEL_PRINT
LIN {X -2.7876,Y -115.7905,Z 117,A -95.3048,B 24.9573,C -1.5092,E1 24.9955,E2 181.3692} C_DIS
LIN {X -5.6832,Y -115.6848,Z 117,A -96.7368,B 24.9573,C -1.5092,E1 24.9915,E2 182.8017} C_DIS
LIN {X -8.4658,Y -115.5142,Z 117,A -98.116,B 24.9573,C -1.5092,E1 24.9876,E2 184.1814} C_DIS
LIN {X -11.1945,Y -115.2812,Z 117,A -99.4758,B 24.9573,C -1.509,E1 24.9839,E2 185.5422} C_DIS
LIN {X -14.1236,Y -114.9597,Z 117,A -100.9264,B 24.9573,C -1.5095,E1 24.9798,E2 186.9926} C_DIS
LIN {X -16.9406,Y -114.5784,Z 117,A -102.3368,B 24.9573,C -1.5096,E1 24.9759,E2 188.4038} C_DIS
LIN {X -19.7474,Y -114.1282,Z 117,A -103.7414,B 24.9573,C -1.5101,E1 24.9721,E2 189.8086} C_DIS
LIN {X -22.5423,Y -113.6092,Z 117,A -105.1516,B 24.9573,C -1.5105,E1 24.9682,E2 191.2194} C_DIS
LIN {X -25.3773,Y -113.0101,Z 117,A -106.5853,B 24.9573,C -1.5111,E1 24.9643,E2 192.6534} C_DIS
LIN {X -28.143,Y -112.3532,Z 117,A -107.9932,B 24.9572,C -1.5118,E1 24.9605,E2 194.0615} C_DIS
LIN {X -30.8918,Y -111.6287,Z 117,A -109.4015,B 24.9572,C -1.5126,E1 24.9567,E2 195.4701} C_DIS
LIN {X -33.1661,Y -110.9723,Z 117,A -110.6229,B 24.9572,C -1.5113,E1 24.9534,E2 196.6967} C_DIS
LIN {X -36.2798,Y -109.9954,Z 117,A -112.1912,B 24.957,C -1.5145,E1 24.9492,E2 198.2602} C_DIS
LIN {X -38.9682,Y -109.0719,Z 117,A -113.5996,B 24.957,C -1.5156,E1 24.9455,E2 199.6687} C_DIS
LIN {X -41.6333,Y -108.0827,Z 117,A -115.0039,B 24.9569,C -1.517,E1 24.9418,E2 201.0726} C_DIS
LIN {X -44.2732,Y -107.0284,Z 117,A -116.4185,B 24.9569,C -1.5181,E1 24.9382,E2 202.4878} C_DIS
LIN {X -46.8865,Y -105.9097,Z 117,A -117.829,B 24.9567,C -1.5194,E1 24.9346,E2 203.8984} C_DIS
LIN {X -49.4715,Y -104.7271,Z 117,A -119.2379,B 24.9567,C -1.5209,E1 24.931,E2 205.3073} C_DIS
LIN {X -52.0759,Y -103.4571,Z 117,A -120.6749,B 24.9566,C -1.5226,E1 24.9274,E2 206.7443} C_DIS
LIN {X -54.5992,Y -102.1479,Z 117,A -122.0852,B 24.9565,C -1.5242,E1 24.9239,E2 208.1545} C_DIS
LIN {X -57.0417,Y -100.804,Z 117,A -123.4682,B 24.9564,C -1.526,E1 24.9205,E2 209.5373} C_DIS
LIN {X -59.4984,Y -99.3738,Z 117,A -124.8788,B 24.9563,C -1.5278,E1 24.9172,E2 210.9477} C_DIS
LIN {X -61.9192,Y -97.8837,Z 117,A -126.2899,B 24.9562,C -1.5298,E1 24.9138,E2 212.3586} C_DIS
LIN {X -63.9596,Y -96.5609,Z 117,A -127.5439,B 24.9562,C -1.5296,E1 24.9109,E2 213.6173} C_DIS
LIN {X -66.229,Y -95.0185,Z 117,A -128.9262,B 24.9561,C -1.5308,E1 24.9077,E2 215.0014} C_DIS
LIN {X -68.9965,Y -93.031,Z 117,A -130.5511,B 24.9558,C -1.5362,E1 24.904,E2 216.6191} C_DIS
LIN {X -70.8835,Y -91.5989,Z 117,A -131.7809,B 24.9558,C -1.5359,E1 24.9013,E2 217.8541} C_DIS
LIN {X -73.4355,Y -89.568,Z 117,A -133.3473,B 24.9555,C -1.5409,E1 24.8979,E2 219.4145} C_DIS
LIN {X -75.6115,Y -87.7388,Z 117,A -134.7595,B 24.9554,C -1.5433,E1 24.8949,E2 220.8264} C_DIS
LIN {X -77.3629,Y -86.1961,Z 117,A -135.9912,B 24.9554,C -1.5425,E1 24.8923,E2 222.065} C_DIS
LIN {X -79.8656,Y -83.8854,Z 117,A -137.6115,B 24.9551,C -1.5486,E1 24.889,E2 223.6774} C_DIS
LIN {X -81.9002,Y -81.9002,Z 117,A -139.0241,B 24.9549,C -1.5513,E1 24.8862,E2 225.0894} C_DIS
LIN {X -83.8473,Y -79.9051,Z 117,A -140.4101,B 24.9548,C -1.554,E1 24.8835,E2 226.4749} C_DIS
LIN {X -85.7831,Y -77.8233,Z 117,A -141.8228,B 24.9546,C -1.5569,E1 24.8809,E2 227.887} C_DIS
LIN {X -87.7032,Y -75.6533,Z 117,A -143.2634,B 24.9544,C -1.5599,E1 24.8782,E2 229.327} C_DIS
LIN {X -90.4284,Y -72.3739,Z 117,A -145.3835,B 24.9541,C -1.5645,E1 24.8745,E2 231.4461} C_DIS
LIN {X -92.1438,Y -70.1764,Z 117,A -146.7699,B 24.954,C -1.5675,E1 24.8721,E2 232.8318} C_DIS
LIN {X -93.8382,Y -67.8939,Z 117,A -148.1766,B 24.9538,C -1.571,E1 24.8698,E2 234.237} C_DIS
LIN {X -95.4762,Y -65.5706,Z 117,A -149.5988,B 24.9536,C -1.5739,E1 24.8675,E2 235.6593} C_DIS
LIN {X -97.0566,Y -63.2077,Z 117,A -151.0127,B 24.9534,C -1.5772,E1 24.8653,E2 237.0723} C_DIS
LIN {X -98.6077,Y -60.7603,Z 117,A -152.4537,B 24.9532,C -1.5807,E1 24.8632,E2 238.5124} C_DIS
LIN {X -100.0691,Y -58.322,Z 117,A -153.8679,B 24.953,C -1.5842,E1 24.8612,E2 239.9257} C_DIS
LIN {X -101.4702,Y -55.8486,Z 117,A -155.2824,B 24.9528,C -1.5877,E1 24.8593,E2 241.3392} C_DIS
LIN {X -102.7847,Y -53.3902,Z 117,A -156.6698,B 24.9526,C -1.5912,E1 24.8575,E2 242.7257} C_DIS
LIN {X -104.064,Y -50.8516,Z 117,A -158.0854,B 24.9523,C -1.5947,E1 24.8557,E2 244.1404} C_DIS
LIN {X -105.3038,Y -48.2327,Z 117,A -159.5267,B 24.9521,C -1.5985,E1 24.854,E2 245.5806} C_DIS
LIN {X -106.4558,Y -45.6339,Z 117,A -160.9419,B 24.9519,C -1.6022,E1 24.8524,E2 246.9949} C_DIS
LIN {X -107.3287,Y -43.5356,Z 117,A -162.1469,B 24.9519,C -1.6022,E1 24.8512,E2 248.2064} C_DIS
LIN {X -108.5667,Y -40.3554,Z 117,A -163.7721,B 24.9514,C -1.6097,E1 24.8495,E2 249.8229} C_DIS
LIN {X -109.5243,Y -37.6788,Z 117,A -165.1875,B 24.9512,C -1.6136,E1 24.8482,E2 251.2372} C_DIS
LIN {X -110.416,Y -34.9796,Z 117,A -166.6031,B 24.951,C -1.6175,E1 24.847,E2 252.6517} C_DIS
LIN {X -111.2256,Y -32.312,Z 117,A -167.9912,B 24.9507,C -1.6213,E1 24.8459,E2 254.0385} C_DIS
LIN {X -111.9851,Y -29.5726,Z 117,A -169.3984,B 24.9505,C -1.6256,E1 24.8449,E2 255.4437} C_DIS
LIN {X -112.6771,Y -26.8155,Z 117,A -170.8235,B 24.9503,C -1.6292,E1 24.8439,E2 256.8686} C_DIS
LIN {X -113.3013,Y -24.0422,Z 117,A -172.2382,B 24.95,C -1.6333,E1 24.8431,E2 258.2819} C_DIS
LIN {X -113.8675,Y -21.2005,Z 117,A -173.6813,B 24.9498,C -1.6374,E1 24.8423,E2 259.7238} C_DIS
LIN {X -114.3535,Y -18.3996,Z 117,A -175.0973,B 24.9495,C -1.6414,E1 24.8417,E2 261.1384} C_DIS
LIN {X -114.7706,Y -15.5877,Z 117,A -176.5132,B 24.9493,C -1.6455,E1 24.8411,E2 262.5531} C_DIS
LIN {X -115.1186,Y -12.7664,Z 117,A -177.9294,B 24.949,C -1.6496,E1 24.8407,E2 263.9679} C_DIS
LIN {X -115.3922,Y -9.9921,Z 117,A -179.3189,B 24.9488,C -1.6537,E1 24.8403,E2 265.3562} C_DIS
LIN {X -115.6064,Y -7.1024,Z 117,A 179.2387,B 24.9485,C -1.6579,E1 24.84,E2 266.7971} C_DIS
LIN {X -115.7435,Y -4.318,Z 117,A 177.8554,B 24.9482,C -1.6622,E1 24.8399,E2 268.1785} C_DIS
LIN {X -115.8156,Y -1.4213,Z 117,A 176.3626,B 24.9481,C -1.6645,E1 24.8398,E2 269.6749} C_DIS
LIN {X -115.8163,Y 1.3214,Z 117,A 175.0356,B 24.9477,C -1.6701,E1 24.8398,E2 270.9965} C_DIS
LIN {X -115.7459,Y 4.2632,Z 117,A 173.5739,B 24.9475,C -1.6746,E1 24.8399,E2 272.4563} C_DIS
LIN {X -115.6064,Y 7.1024,Z 117,A 172.1581,B 24.9472,C -1.6788,E1 24.8401,E2 273.8707} C_DIS
LIN {X -115.3973,Y 9.9374,Z 117,A 170.7416,B 24.9469,C -1.6829,E1 24.8405,E2 275.2857} C_DIS
LIN {X -115.1243,Y 12.7118,Z 117,A 169.3529,B 24.9467,C -1.687,E1 24.8409,E2 276.673} C_DIS
LIN {X -114.8059,Y 15.316,Z 117,A 168.0294,B 24.9465,C -1.6902,E1 24.8413,E2 277.9967} C_DIS
LIN {X -114.3619,Y 18.3454,Z 117,A 166.5208,B 24.9461,C -1.6954,E1 24.842,E2 279.502} C_DIS
LIN {X -113.9114,Y 20.9565,Z 117,A 165.184,B 24.9459,C -1.6986,E1 24.8426,E2 280.8391} C_DIS
LIN {X -113.313,Y 23.9885,Z 117,A 163.6612,B 24.9456,C -1.7037,E1 24.8435,E2 282.3586} C_DIS
LIN {X -112.6901,Y 26.7622,Z 117,A 162.2453,B 24.9453,C -1.7079,E1 24.8444,E2 283.773} C_DIS
LIN {X -112.0131,Y 29.4665,Z 117,A 160.8555,B 24.9451,C -1.7119,E1 24.8453,E2 285.1614} C_DIS
LIN {X -111.2412,Y 32.2594,Z 117,A 159.4132,B 24.9448,C -1.716,E1 24.8464,E2 286.602} C_DIS
LIN {X -110.4323,Y 34.9272,Z 117,A 158.0246,B 24.9446,C -1.72,E1 24.8476,E2 287.9891} C_DIS
LIN {X -109.5243,Y 37.6788,Z 117,A 156.5816,B 24.9443,C -1.7241,E1 24.8488,E2 289.4306} C_DIS
LIN {X -108.5855,Y 40.3038,Z 117,A 155.1952,B 24.944,C -1.7282,E1 24.8502,E2 290.8152} C_DIS
LIN {X -107.5436,Y 43.0076,Z 117,A 153.7502,B 24.9438,C -1.7321,E1 24.8516,E2 292.2588} C_DIS
LIN {X -106.4558,Y 45.6339,Z 117,A 152.3344,B 24.9435,C -1.7361,E1 24.8532,E2 293.6731} C_DIS
LIN {X -105.3038,Y 48.2327,Z 117,A 150.9192,B 24.9433,C -1.74,E1 24.8548,E2 295.0867} C_DIS
LIN {X -104.0884,Y 50.8024,Z 117,A 149.5035,B 24.943,C -1.7439,E1 24.8565,E2 296.5009} C_DIS
LIN {X -102.8103,Y 53.3416,Z 117,A 148.0883,B 24.9428,C -1.7477,E1 24.8583,E2 297.9146} C_DIS
LIN {X -101.4702,Y 55.8486,Z 117,A 146.6731,B 24.9425,C -1.7515,E1 24.8602,E2 299.3282} C_DIS
LIN {X -100.0691,Y 58.322,Z 117,A 145.2578,B 24.9423,C -1.7552,E1 24.8621,E2 300.742} C_DIS
LIN {X -98.6362,Y 60.7133,Z 117,A 143.8778,B 24.942,C -1.7592,E1 24.8641,E2 302.1197} C_DIS
LIN {X -97.0868,Y 63.1619,Z 117,A 142.428,B 24.9418,C -1.7626,E1 24.8663,E2 303.5687} C_DIS
LIN {X -95.5383,Y 65.4801,Z 117,A 141.0396,B 24.9415,C -1.7661,E1 24.8685,E2 304.9556} C_DIS
LIN {X -94.0448,Y 67.6056,Z 117,A 139.7279,B 24.9414,C -1.7686,E1 24.8706,E2 306.2678} C_DIS
LIN {X -92.2103,Y 70.089,Z 117,A 138.2105,B 24.9411,C -1.7731,E1 24.8731,E2 307.7818} C_DIS
LIN {X -90.6204,Y 72.131,Z 117,A 136.9024,B 24.9409,C -1.7754,E1 24.8754,E2 309.0904} C_DIS
Enddeposition()
END
